RV571.GetState_AI();
RV571(bSetStatusOnAutomatic := bSetStatusOn_RV500,
	fSetPointAutomatic := fSetPoint,
	bAlgorithmPermission := bAlgorithmPermission,
	fTemperatureExternal := fMeanHallTemperature,
	nControlModeAutomatic := nControlMode_RV500);
RV571.SetState_AO();

RV572.GetState_AI();
RV572(bSetStatusOnAutomatic := bSetStatusOn_RV500,
	fSetPointAutomatic := fSetPoint,
	bAlgorithmPermission := bAlgorithmPermission,
	fTemperatureExternal := fMeanHallTemperature,
	nControlModeAutomatic := nControlMode_RV500);
RV572.SetState_AO();

RV573.GetState_AI();
RV573(bSetStatusOnAutomatic := bSetStatusOn_RV500,
	fSetPointAutomatic := fSetPoint,
	bAlgorithmPermission := bAlgorithmPermission,
	fTemperatureExternal := fMeanHallTemperature,
	nControlModeAutomatic := nControlMode_RV500);
RV573.SetState_AO();

//sensors
PS500();
PS500.GetState_AI();
TS541();
TS541.GetState_AI();
TS542();
TS542.GetState_AI();
TS543();
TS543.GetState_AI();
TS551();
TS551.GetState_AI();
TS552();
TS552.GetState_AI();
TS553();
TS553.GetState_AI();
TS561();
TS561.GetState_AI();
TS562();
TS562.GetState_AI();
TS563();
TS563.GetState_AI();
TS571();
TS571.GetState_AI();
TS572();
TS572.GetState_AI();
TS573();
TS573.GetState_AI();

WMZ405(aHeatCounterTelegramm := aTelegramm_WMZ405);

METHOD CalculateAverageTemperature : REAL
VAR_INPUT
	fActualTemperature : REAL;
END_VAR
VAR_OUTPUT
	fMeanTemperature : REAL;
END_VAR
VAR_INST
	fTemperature_init : REAL;
	fMinutes_Moving_Average : UINT := 2;
	
	stParameters_Average_Temperature : ST_CTRL_MOVING_AVERAGE_PARAMS;
	aHallTemperatureBuffer 				: ARRAY [1..360] OF FLOAT := [360(15)];
END_VAR
//fTemperature_init := 

stParameters_Average_Temperature.tCtrlCycleTime := T#1S;
stParameters_Average_Temperature.tTaskCycleTime := GlobalVariables.tTaskCycleTime_MAIN;
stParameters_Average_Temperature.nSamplesToFilter := fMinutes_Moving_Average*60; (* 1min= 60 sec*)
stParameters_Average_Temperature.pWorkArray_ADR := ADR(aHallTemperatureBuffer);
stParameters_Average_Temperature.nWorkArray_SIZEOF := SIZEOF(aHallTemperatureBuffer);

Moving_Average_Hall_Temperature(
	fIn := fActualTemperature,
	fManSyncValue := 15,
	bSync := FALSE,
	eMode := 2,
	bHold := FALSE,
	stParams := stParameters_Average_Temperature);
fMeanTemperature := LREAL_TO_REAL(Moving_Average_Hall_Temperature.fOut);
END_METHOD

METHOD PROTECTED  CheckError : BOOL
VAR_INPUT
END_VAR
VAR_OUTPUT
	bError : BOOL;
END_VAR
VAR
	bError_PU405 : BOOL;
	bError_PU500 : BOOL;
END_VAR
//check pumps for errors
bError_PU405 := PU405.bError;
bError_PU500 := PU500.bError;

bError := bError_PU405 OR bError_PU500;
END_METHOD

METHOD PRIVATE LocalControl : BOOL
VAR_INPUT
END_VAR
VAR
END_VAR
CharacteristicCurve_Parameters.fAmbientTempMax := localDefaultParameters.aLimitsAmbientTemperature[2];
CharacteristicCurve_Parameters.fAmbientTempMin := localDefaultParameters.aLimitsAmbientTemperature[1];
CharacteristicCurve_Parameters.fForeRunTempMax := localDefaultParameters.aLimitsFeedTemperature[1];
CharacteristicCurve_Parameters.fForeRunTempMin := localDefaultParameters.aLimitsFeedTemperature[2];
CharacteristicCurve_Parameters.tCtrlCycleTime := GlobalVariables.tCtrlCycleTime_MAIN;
CharacteristicCurve_Parameters.tTaskCycleTime := GlobalVariables.tTaskCycleTime_MAIN;

CharacteristicCurve(fAmbientTemperature := stAmbientState.fOutsideTemperature,
	fOffsetTemperature := 0,
	bLimitFlowTemp := TRUE,
	stParams := CharacteristicCurve_Parameters);
fSetPoint_RV500 := LREAL_TO_REAL(CharacteristicCurve.fOut);
	
IF bHeatingMode THEN
	nControlMode_RV500 := 1;
ELSE
	nControlMode_RV500 := 2;	
END_IF
END_METHOD

METHOD PROTECTED  Operational : BOOL
VAR_INPUT
END_VAR
VAR_OUTPUT
	bSwitchToWorking : BOOL := FALSE;
END_VAR
bSetStatusOn_RV500 := TRUE;
bSetStatusOn_PU405 := TRUE;
bSetStatusOn_PU500 := TRUE;

IF PU405.bStatusOn AND PU500.bStatusOn THEN
	bSwitchToWorking := TRUE;
END_IF
END_METHOD

METHOD PROTECTED  RampDown : BOOL
VAR_INPUT
END_VAR
VAR_OUTPUT
	bRampDownFinished : BOOL := FALSE;
END_VAR
bSetStatusOn_PU405 := FALSE;
bSetStatusOn_PU500 := FALSE;
bSetStatusOn_RV500 := FALSE;
bSetStatusOn_SV_HNLT := FALSE;
bSetStatusOn_SV_CN := FALSE;
	
IF SV_HNLT.localState.nPosition=2 AND SV_HNLT.localState.nPosition=2 AND SV_CN.localState.nPosition=2 AND SV_CN.localState.nPosition=2 THEN
	bRampDownFinished := TRUE;		
END_IF
END_METHOD

METHOD PROTECTED  RampUp : BOOL
VAR_INPUT
END_VAR
VAR_OUTPUT
	bRampUpFinished : BOOL := FALSE;
END_VAR
IF bHeatingMode THEN
	bSetStatusOn_SV_HNLT := TRUE;
	bSetStatusOn_SV_CN := FALSE;
	IF SV_HNLT.localState.nPosition=3 AND SV_HNLT.localState.nPosition=3 AND SV_CN.localState.nPosition=2 AND SV_CN.localState.nPosition=2 THEN
		bRampUpFinished := TRUE;		
	END_IF	
ELSE
	bSetStatusOn_SV_HNLT := FALSE;
	bSetStatusOn_SV_CN := TRUE;
	IF SV_HNLT.localState.nPosition=2 AND SV_HNLT.localState.nPosition=2 AND SV_CN.localState.nPosition=3 AND SV_CN.localState.nPosition=3 THEN
		bRampUpFinished := TRUE;		
	END_IF	
END_IF
END_METHOD

METHOD PRIVATE SelectLocalControlMode : BOOL
VAR_INPUT
END_VAR
IF control.bManualModeActivated THEN
	bHeatingMode := localSetParameters.bHeatingModeManual;
ELSIF control.bAlgorithmModeActivated AND bAlgorithmPermission THEN
	bHeatingMode := localSetParameters.bHeatingModeAlgorithm;
ELSE
	bHeatingMode := bHeatingModeAutomatic;
END_IF
END_METHOD

METHOD PROTECTED   SetSetPointLimits : BOOL
VAR_INPUT
END_VAR
aSetPointLimits[1] := localDefaultParameters.aSetPointLimitsTemperature[1];
aSetPointLimits[2] := localDefaultParameters.aSetPointLimitsTemperature[2];
END_METHOD

METHOD PROTECTED  SetState : BOOL
VAR_INPUT
END_VAR
VAR_OUTPUT
END_VAR
fOperatingPoint := stAmbientState.fHallTemperature;

controlState.bStatusOn := bSetStatusOn;
setPointState.aSetPointLimits := aSetPointLimits;
setPointState.fSetPoint := fSetPoint;
setPointState.fOperatingPoint := fOperatingPoint;
setPointState.sSetPointUnit := 'degreeC';
setPointState.sOperatingPointUnit := 'degreeC';
END_METHOD

METHOD PRIVATE SwitchMode : BOOL
VAR_INPUT
	bSwitchToHeating : BOOL; //if false switch to cooling
END_VAR
VAR_OUTPUT
	bFinishedSwitchMode : BOOL := FALSE;
END_VAR
VAR_INST
	bRampDownFinished : BOOL := FALSE;
END_VAR
//check system state
IF bRampDownFinished THEN
	IF bSwitchToHeating THEN
		//close valve in cooling network
		bSetStatusOn_SV_CN := FALSE;	
		IF SV_CN.localState.nPosition=2 AND SV_CN.localState.nPosition=2 THEN
			bSetStatusOn_SV_HNLT := TRUE;	
		END_IF

		IF SV_HNLT.localState.nPosition=3 AND SV_HNLT.localState.nPosition=3 THEN
			//reset instant variable and switch on pump
			bRampDownFinished := FALSE;			
			bFinishedSwitchMode := TRUE;
			bSetStatusOn_PU405 := TRUE;
		END_IF
		
	ELSE
		//close valve in heating network
		bSetStatusOn_SV_HNLT := FALSE;
		//wait until valves in heating network are closed before opening valves in cooling network
		IF SV_HNLT.localState.nPosition=2 AND SV_HNLT.localState.nPosition=2 THEN
			bSetStatusOn_SV_CN := TRUE;
		END_IF
		IF SV_CN.localState.nPosition=3 AND SV_CN.localState.nPosition=3 THEN
			//reset instant variable and switch on pump
			bRampDownFinished := FALSE;			
			bFinishedSwitchMode := TRUE;
			bSetStatusOn_PU405 := TRUE;	
		END_IF
	END_IF
ELSE
	bSetStatusOn_PU405 := FALSE;
	IF NOT PU405.bStatusOn THEN
		bRampDownFinished := TRUE;
	END_IF
END_IF
END_METHOD

METHOD PROTECTED  Working : BOOL
VAR_INPUT
END_VAR
VAR_OUTPUT
	bSwitchToOperational : BOOL := FALSE;
END_VAR
//empty method
END_METHOD

END_FUNCTION_BLOCK

// ---- POUs/04 Systems/LinkageSystems/FB_UnderfloorHeatingSystem.TcPOU
FUNCTION_BLOCK FB_UnderfloorHeatingSystem EXTENDS FB_SystemContinous
VAR_INPUT
	bHeatingModeAutomatic : BOOL; //control mode: 0 = heating mode, 1 = cooling mode
	stAmbientState : ST_AmbientState;
END_VAR
VAR_OUTPUT
END_VAR
VAR
	{attribute 'OPC.UA.DA' := '1'}
	localSetParameters : ST_UnderfloorHeatingSetParameters;

	//default parameters
	localDefaultParameters : ST_UnderfloorHeatingDefaultParameters;	
	
	//pumps
	stPU425DefaultParameters : ST_PumpGrundfosMagna3DefaultParameters;
	PU425 : FB_PumpGrundfosMagna3 := (ST_DefaultParameters := stPU425DefaultParameters);	
	
	//valves
	stSV423DefaultParameters : ST_DiscreteValveDefaultParameters := (nFeedback := 3);
	stSV424DefaultParameters : ST_DiscreteValveDefaultParameters := (nFeedback := 3);
	stRV425DefaultParameters : ST_MixingValveDefaultParameters := (bFeedbackSignal := FALSE, tTaskCycleTime := GlobalVariables.tTaskCycleTime_MAIN, tCtrlCycleTime := GlobalVariables.tCtrlCycleTime_MAIN);	
	
	SV423 : FB_DiscreteValve := (ST_DefaultParameters := stSV423DefaultParameters); 
	SV424 : FB_DiscreteValve := (ST_DefaultParameters := stSV424DefaultParameters);
	RV425 : FB_MixingValve := (ST_DefaultParameters := stRV425DefaultParameters);
	WMZ425 : FB_MollineEHeatCounter;
	
	//internal variables
	bHeatingMode 			: BOOL;
	bSetStatusOn_PU425 		: BOOL;
	bSetStatusOn_SV423		: BOOL;
	bSetStatusOn_SV424		: BOOL;
	bSetStatusOn_RV425 		: BOOL;
	fSetPoint_Internal 		: REAL;
	nControlMode_RV425 		: E_MixingValveControlMode; 	
	
	//characteristic curves and controllers
	CharacteristicCurve 			: FB_CTRL_FLOW_TEMP_SETPOINT_GEN;
	CharacteristicCurve_Parameters	: ST_CTRL_FLOW_TEMP_SETPOINT_GEN_PARAMS;
	
	//triggers
	SwitchToHeating : R_TRIG;
	SwitchToCooling : F_TRIG;
	bFinishedSwitchMode : BOOL := TRUE;
END_VAR

//check if heating mode has switched
SelectLocalControlMode();
LocalControl();
fSetPointAutomatic := fSetPoint_Internal;
SwitchToHeating(CLK := bHeatingMode);
SwitchToCooling(CLK := bHeatingMode);

//MAIN must be called before SwitchMode to prevent pump signal chattering (signal is written after SwitchMode function), SwitchMode may only be called if system is on
MAIN();

//disrupt calling SystemFlowControl via MAIN() when mode is switched and call SwitchMode()
IF ((SwitchToHeating.Q OR SwitchToCooling.Q) OR NOT bFinishedSwitchMode) AND bSetStatusOn THEN
	SwitchMode(bSwitchToHeating := bHeatingMode,
		bFinishedSwitchMode => bFinishedSwitchMode);
END_IF;

//pumps
PU425.GetState_Profibus();
PU425(bSetStatusOnAutomatic := bSetStatusOn_PU425,
	fSetPointAutomatic := 100,
	bAlgorithmPermission := bAlgorithmPermission,
	nControlModeAutomatic := 0);
PU425.SetState_Profibus();

//valves in thermal networks
RV425.GetState_AI();
RV425(bSetStatusOnAutomatic := bSetStatusOn_RV425,
	fSetPointAutomatic := fSetPoint_Internal,
	bAlgorithmPermission := bAlgorithmPermission,
	fTemperatureExternal := PU425.fTemperatureInternal,
	fThermalPowerExternal := WMZ425.fHeatFlowRate,
	nControlModeAutomatic := nControlMode_RV425);
RV425.SetState_AO();

SV423.GetState_BI();
SV423(bSetStatusOnAutomatic := bSetStatusOn_SV423,
	bAlgorithmPermission := bAlgorithmPermission);
SV423.SetState_BO();

SV424.GetState_BI();
SV424(bSetStatusOnAutomatic := bSetStatusOn_SV423,
	bAlgorithmPermission := bAlgorithmPermission);
SV424.SetState_BO();

WMZ425(aHeatCounterTelegramm := aTelegramm_WMZ425);

METHOD PROTECTED  CheckError : BOOL
VAR_INPUT
END_VAR
VAR_OUTPUT
	bError : BOOL;
END_VAR
VAR
END_VAR
//check pumps for errors
bError :=  PU425.bError;
END_METHOD

METHOD PRIVATE LocalControl : BOOL
VAR_INPUT
END_VAR
VAR
END_VAR
CharacteristicCurve_Parameters.fAmbientTempMax := localDefaultParameters.aLimitsAmbientTemperature[2];
CharacteristicCurve_Parameters.fAmbientTempMin := localDefaultParameters.aLimitsAmbientTemperature[1];
CharacteristicCurve_Parameters.fForeRunTempMax := localDefaultParameters.aLimitsFeedTemperature[1];
CharacteristicCurve_Parameters.fForeRunTempMin := localDefaultParameters.aLimitsFeedTemperature[2];
CharacteristicCurve_Parameters.tCtrlCycleTime := GlobalVariables.tCtrlCycleTime_MAIN;
CharacteristicCurve_Parameters.tTaskCycleTime := GlobalVariables.tTaskCycleTime_MAIN;

CharacteristicCurve(fAmbientTemperature := stAmbientState.fOutsideTemperature,
	fOffsetTemperature := 0,
	bLimitFlowTemp := TRUE,
	stParams := CharacteristicCurve_Parameters);
fSetPoint_Internal := LREAL_TO_REAL(CharacteristicCurve.fOut);
	
IF bHeatingMode THEN
	nControlMode_RV425 := 1;
ELSE
	nControlMode_RV425 := 2;	
END_IF
END_METHOD

METHOD PROTECTED  Operational : BOOL
VAR_INPUT
END_VAR
VAR_OUTPUT
	bSwitchToWorking : BOOL := FALSE;
END_VAR
bSetStatusOn_RV425 := TRUE;
bSetStatusOn_PU425 := TRUE;

IF PU425.bStatusOn THEN
	bSwitchToWorking := TRUE;
END_IF
END_METHOD

METHOD PROTECTED  RampDown : BOOL
VAR_INPUT
END_VAR
VAR_OUTPUT
	bRampDownFinished : BOOL := FALSE;
END_VAR
bSetStatusOn_PU425 := FALSE;
bSetStatusOn_RV425 := FALSE;
	
IF PU425.bStatusOn THEN
	bRampDownFinished := TRUE;		
END_IF
END_METHOD

METHOD PROTECTED  RampUp : BOOL
VAR_INPUT
END_VAR
VAR_OUTPUT
	bRampUpFinished : BOOL := FALSE;
END_VAR
IF bHeatingMode THEN
	//bSetStatusOn_SV423 := FALSE;
	//bSetStatusOn_SV424 := FALSE;
	IF SV423.localState.nPosition=3 AND SV424.localState.nPosition=3 THEN
		bRampUpFinished := TRUE;		
	END_IF	
ELSE
	//bSetStatusOn_SV423 := TRUE;
	//bSetStatusOn_SV424 := TRUE;
	IF SV423.localState.nPosition=2 AND SV424.localState.nPosition=2 THEN
		bRampUpFinished := TRUE;		
	END_IF	
END_IF
END_METHOD

METHOD PRIVATE SelectLocalControlMode : BOOL
VAR_INPUT
END_VAR
IF control.bManualModeActivated THEN
	bHeatingMode := localSetParameters.bHeatingModeManual;
ELSIF control.bAlgorithmModeActivated AND bAlgorithmPermission THEN
	bHeatingMode := localSetParameters.bHeatingModeAlgorithm;
ELSE
	bHeatingMode := bHeatingModeAutomatic;
END_IF
END_METHOD

METHOD PROTECTED   SetSetPointLimits : BOOL
VAR_INPUT
END_VAR
aSetPointLimits[1] := localDefaultParameters.aSetPointLimitsTemperature[1];
aSetPointLimits[2] := localDefaultParameters.aSetPointLimitsTemperature[2];
END_METHOD

METHOD PROTECTED  SetState : BOOL
VAR_INPUT
END_VAR
VAR_OUTPUT
END_VAR
fOperatingPoint := PU425.fTemperatureInternal;

controlState.bStatusOn := bSetStatusOn;
setPointState.aSetPointLimits := aSetPointLimits;
setPointState.fSetPoint := fSetPoint;
setPointState.fOperatingPoint := fOperatingPoint;
setPointState.sSetPointUnit := 'degreeC';
setPointState.sOperatingPointUnit := 'degreeC';
END_METHOD

METHOD PRIVATE SwitchMode : BOOL
VAR_INPUT
	bSwitchToHeating : BOOL; //if false switch to cooling
END_VAR
VAR_OUTPUT
	bFinishedSwitchMode : BOOL := FALSE;
END_VAR
VAR_INST
	bRampDownFinished : BOOL := FALSE;
END_VAR
//check system state
IF bRampDownFinished THEN
	IF bSwitchToHeating THEN
		//false - valve connects heating network
		bSetStatusOn_SV423 := FALSE;
		bSetStatusOn_SV424 := FALSE;	

		IF SV423.localState.nPosition=3 AND SV424.localState.nPosition=3 THEN
			//reset instant variable and switch on pump
			bRampDownFinished := FALSE;			
			bFinishedSwitchMode := TRUE;
			bSetStatusOn_PU425 := TRUE;
		END_IF
		
	ELSE
		//true - connects cooling network
		bSetStatusOn_SV423 := TRUE;
		bSetStatusOn_SV424 := TRUE;	

		IF SV423.localState.nPosition=2 AND SV424.localState.nPosition=2 THEN
			//reset instant variable and switch on pump
			bRampDownFinished := FALSE;			
			bFinishedSwitchMode := TRUE;
			bSetStatusOn_PU425 := TRUE;
		END_IF
	END_IF
ELSE
	bSetStatusOn_PU425 := FALSE;
	IF NOT PU425.bStatusOn THEN
		bRampDownFinished := TRUE;
	END_IF
END_IF
END_METHOD

METHOD PROTECTED  Working : BOOL
VAR_INPUT
END_VAR
VAR_OUTPUT
	bSwitchToOperational : BOOL := FALSE;
END_VAR
//empty method
END_METHOD

END_FUNCTION_BLOCK

// ---- POUs/05 Thermal Networks/FB_HnhtCnLinkage.TcPOU
FUNCTION_BLOCK FB_HnhtCnLinkage
VAR_INPUT	
	//control struct for hnht cn linkage
	controlAutomatic : ST_HnhtCnLinkageControl;
END_VAR
VAR_OUTPUT
END_VAR
VAR
	//systems
	VentilationSystem : FB_VentilationSystem;
	
	//internal variables
	bAlgorithmPermission : BOOL;
	
	//PCM Supply System
	PCMSupplySystem : FB_PCMSupplySystem;
END_VAR

bAlgorithmPermission := controlAutomatic.bAlgorithmPermission_HNHT AND controlAutomatic.bAlgorithmPermission_CN;

//ventilation system has its own controller, only valves are controlled
VentilationSystem(bSetStatusOnAutomatic := TRUE,
	fSetPointAutomatic := 0,
	bAlgorithmPermission := bAlgorithmPermission,
	bHeatingModeAutomatic := controlAutomatic.bHeatingMode);

PCMSupplySystem(bSetStatusOnAutomatic := TRUE, 
	bAlgorithmPermission := bAlgorithmPermission,
	fSetPointAutomatic := 9);

END_FUNCTION_BLOCK

// ---- POUs/04 Systems/LinkageSystems/FB_VentilationSystem.TcPOU
FUNCTION_BLOCK FB_VentilationSystem EXTENDS FB_SystemContinous
VAR_INPUT
	bHeatingModeAutomatic : BOOL; //control mode: 0 = heating mode, 1 = cooling mode
END_VAR
VAR_OUTPUT
END_VAR
VAR
	{attribute 'OPC.UA.DA' := '1'}
	localSetParameters : ST_VentilationSetParameters;
	
	localDefaultParameters : ST_VentilationDefaultParameters;
	
	//valves
	stSV453DefaultParameters : ST_DiscreteValveDefaultParameters := (nFeedback := 3);
	stSV454DefaultParameters : ST_DiscreteValveDefaultParameters := (nFeedback := 3);
	SV453 : FB_DiscreteValve := (ST_DefaultParameters := stSV453DefaultParameters);
	SV454 : FB_DiscreteValve := (ST_DefaultParameters := stSV454DefaultParameters);
	
	//pump (pump is just read)
	stPU455DefaultParameters : ST_PumpGrundfosMagna3DefaultParameters := (tTaskCycleTime := GlobalVariables.tTaskCycleTime_MAIN, tCtrlCycleTime := GlobalVariables.tCtrlCycleTime_MAIN);
	PU455 : FB_PumpGrundfosMagna3 := (ST_DefaultParameters := stPU455DefaultParameters);
	
	WMZ455 : FB_MollineEHeatCounter;
	
	//ventilation 
	//Ventilation : FB_Ventilation; //commented out for merge in dev, as modbus write needs to be deactivated before bugs are fixed
	
	//electricity meter
	EM45x : FB_JanitzaSensor;
	
	
	
	bHeatingMode 			: BOOL;
	bSetStatusOn_SV453		: BOOL;
	bSetStatusOn_SV454		: BOOL;
END_VAR

SelectLocalControlMode();
MAIN();
(* Ventilation.GetState();
Ventilation(
	fSetPointAutomatic := fSetPoint,
	bSetStatusOnAutomatic := FALSE,
	bAlgorithmPermission := bAlgorithmPermission,
	sIPAddress := GlobalVariables.sIP_Ventilation);
Ventilation.SetState();
EM45x(
	sIPAddress := GlobalVariables.sIP_Janitza_Ventilation);  

*)

IF bHeatingMode THEN
	bSetStatusOn_SV453 := TRUE;
	bSetStatusOn_SV454 := TRUE;
ELSE
	bSetStatusOn_SV453 := FALSE;
	bSetStatusOn_SV454 := FALSE;
END_IF

SV453.GetState_BI();
SV453(bSetStatusOnAutomatic := bSetStatusOn_SV453,
	bAlgorithmPermission := bAlgorithmPermission);
SV453.SetState_BO();

SV454.GetState_BI();
SV454(bSetStatusOnAutomatic := bSetStatusOn_SV454,
	bAlgorithmPermission := bAlgorithmPermission);
SV454.SetState_BO();


	
	
	
	

//PU455 and RV455 is controlled by ventilation unit
PU455.GetState_Profibus();
PU455();

WMZ455(aHeatCounterTelegramm := aTelegramm_WMZ455);

METHOD PROTECTED  CheckError : BOOL
VAR_INPUT
END_VAR
VAR_OUTPUT
	bError : BOOL;
END_VAR
IF (SV453.localState.nPosition = 2 AND SV454.localState.nPosition = 3) OR (SV453.localState.nPosition = 3 AND SV454.localState.nPosition = 2) THEN
	bError := TRUE;
ELSE
	bError := FALSE;
END_IF
END_METHOD

METHOD PROTECTED  Operational : BOOL
VAR_INPUT
END_VAR
VAR_OUTPUT
	bSwitchToWorking : BOOL := FALSE;
END_VAR
//empty
END_METHOD

METHOD PROTECTED  RampDown : BOOL
VAR_INPUT
END_VAR
VAR_OUTPUT
	bRampDownFinished : BOOL := FALSE;
END_VAR
//empty
END_METHOD

METHOD PROTECTED  RampUp : BOOL
VAR_INPUT
END_VAR
VAR_OUTPUT
	bRampUpFinished : BOOL := FALSE;
END_VAR
//empty
END_METHOD

METHOD PRIVATE SelectLocalControlMode : BOOL
VAR_INPUT
END_VAR
IF control.bManualModeActivated THEN
	bHeatingMode := localSetParameters.bHeatingModeManual;
ELSIF control.bAlgorithmModeActivated AND bAlgorithmPermission THEN
	bHeatingMode := localSetParameters.bHeatingModeAlgorithm;
ELSE
	bHeatingMode := bHeatingModeAutomatic;
END_IF
END_METHOD

METHOD PROTECTED   SetSetPointLimits : BOOL
VAR_INPUT
END_VAR
aSetPointLimits[1] := localDefaultParameters.aSetPointLimitsTemperature[1];
aSetPointLimits[2] := localDefaultParameters.aSetPointLimitsTemperature[2];
END_METHOD

METHOD PROTECTED  SetState : BOOL
VAR_INPUT
END_VAR
VAR_OUTPUT
END_VAR
fOperatingPoint := 0;

controlState.bStatusOn := bSetStatusOn;
setPointState.aSetPointLimits := aSetPointLimits;
setPointState.fSetPoint := 0;
setPointState.fOperatingPoint := fOperatingPoint;
setPointState.sSetPointUnit := '-';
setPointState.sOperatingPointUnit := '-';
END_METHOD

METHOD PROTECTED  Working : BOOL
VAR_INPUT
END_VAR
VAR_OUTPUT
	bSwitchToOperational : BOOL := FALSE;
END_VAR
//empty
END_METHOD

END_FUNCTION_BLOCK

// ---- POUs/02 Sensors/FB_JanitzaSensor.TcPOU
FUNCTION_BLOCK FB_JanitzaSensor
VAR_INPUT
	sIPAddress : STRING(15);
END_VAR
VAR_OUTPUT
	fPower : REAL; //measured power in watt
	bError : BOOL; 
	nErrID : UDINT; 
END_VAR
VAR
	
	{attribute 'OPC.UA.DA' := '1'}
	sensorState : ST_JanitzaState;
	//modbus tcp communication
	ModbusReader_19026 : FB_MBReadInputRegs; //read reg 19026 (power (W) ventilation)
	
	//define array to store data from every ModbusReader
	aModbus_19026 : ARRAY [0..1] OF WORD;
	
	//modbus timer
	bReadModbus	: BOOL := FALSE;
	bStartTimer : BOOL;
	Timer : TON;
	
	bAwaitData : BOOL; //mark: Results of this still pending
	aTmp : ARRAY[0..1] OF WORD; //temp. buffer for byte-swap (won't overwrite the original)
	
END_VAR

//Start and check timer for 2s interval
Timer(IN := bStartTimer,
	PT := T#2S);
	
bStartTimer := TRUE;
IF Timer.Q THEN
	bReadModbus := TRUE;
	bStartTimer := FALSE;	
	bAwaitData := TRUE; // we expecting a answer
END_IF

ModbusReader_19026(
	sIPAddr := sIPAddress,
	nTCPPort := 502,
	nUnitID := 32,
	nQuantity := 2,
	nMBAddr := 19026 + 32768,
	cbLength := 4,
	pDestAddr := ADR(aModbus_19026),
	bExecute := bReadModbus,
	tTimeout  := T#20S);
	
bReadModbus := FALSE;
	
bError := ModbusReader_19026.bError;
nErrID := ModbusReader_19026.nErrId; 

IF bAwaitData AND NOT ModbusReader_19026.bBusy AND NOT ModbusReader_19026.bError THEN
	bAwaitData := FALSE; 
    // Byte-Swap for every WORD (51794 = 19026+32768: Word sequence is LE, But the Bytes in the Word are BE)
    aModbus_19026[0] := SHL(aModbus_19026[0] AND 16#00FF, 8) OR SHR(aModbus_19026[0] AND 16#FF00, 8);
    aModbus_19026[1] := SHL(aModbus_19026[1] AND 16#00FF, 8) OR SHR(aModbus_19026[1] AND 16#FF00, 8);
	MEMCPY(ADR(fPower), ADR(aModbus_19026), SIZEOF(fPower));
	bStartTimer := TRUE; 
END_IF

//sensor state
sensorState.fPower := fPower/1000;
sensorState.sPowerUnit := 'kW';

END_FUNCTION_BLOCK

// ---- POUs/04 Systems/CoolingSystems/FB_PCMSupplySystem.TcPOU
FUNCTION_BLOCK FB_PCMSupplySystem EXTENDS FB_SystemContinous
VAR_INPUT
	nControlModeAutomatic : E_PCMSystemControlMode;
	
END_VAR
VAR_OUTPUT
END_VAR
VAR
	
	{attribute 'OPC.UA.DA' := '1'}
	localSetParameters : ST_PCMSystemSetParameters;
	
	//heat meters
	WMZ900 : FB_MollineUltramess403HeatCounter; //pcm storage
	WMZ935 : FB_MollineUltramess403HeatCounter; //chiller
	
	//temperature sensors
	
	TS901 : FB_TemperatureSensor_KL3214;
	TS902 : FB_TemperatureSensor_KL3214;
	TS903 : FB_TemperatureSensor_KL3214;
	TS910 : FB_TemperatureSensor_KL3214;
	TS911 : FB_TemperatureSensor_KL3214;
	TS950 : FB_TemperatureSensor_KL3214;
	TS951 : FB_TemperatureSensor_KL3214;
	
	//valves
	ST_RV950DefaultParameters : ST_MixingValveDefaultParameters := (bFeedbackSignal := FALSE, tTaskCycleTime := GlobalVariables.tTaskCycleTime_MAIN, tCtrlCycleTime := GlobalVariables.tCtrlCycleTime_MAIN);
	RV950 : FB_MixingValve := (ST_DefaultParameters := ST_RV950DefaultParameters);
	
	// pcm chiller
	PCMChiller : FB_PCMChiller;
	
	// PCMStorage
	PCMStorage : FB_PCMStorage;
	
	//internal variables
	nControlMode : E_PCMSystemControlMode;
	
	bSetStatusOn_RV950 : BOOL; 
	
	
END_VAR

SelectLocalControlMode();


WMZ900(aHeatCounterTelegramm := aTelegramm_WMZ900);
WMZ935(aHeatCounterTelegramm := aTelegramm_WMZ935);
	
TS901();
TS901.GetState_AI();
TS902();
TS902.GetState_AI();
TS903();
TS903.GetState_AI();
TS910();
TS910.GetState_AI();
TS911();
TS911.GetState_AI();
TS950();
TS950.GetState_AI();
TS951();
TS951.GetState_AI();

RV950.GetState_AI();
RV950(bSetStatusOnAutomatic := bSetStatusOn_RV950,
	fSetPointAutomatic := 100,
	bAlgorithmPermission := TRUE,
	fTemperatureExternal := TS950.fTemperature,
	nControlModeAutomatic := 0);
RV950.SetState_AO();

PCMChiller.GetState(); 
PCMChiller(bSetStatusOnAutomatic := FALSE, 
	bAlgorithmPermission := bAlgorithmPermission,
	fSetPointAutomatic := fSetPoint);
PCMChiller.SetState();

METHOD PROTECTED  CheckError : BOOL
VAR_INPUT
END_VAR
VAR_OUTPUT
	bError : BOOL;
END_VAR
END_METHOD

METHOD LocalControl : BOOL
VAR_INPUT
	
END_VAR
CASE nControlMode OF
	0: //stand-by
	PCMChiller.bStatusOn := FALSE; 
	 	
	1: //direct cooling 
	PCMChiller.nControlModeAutomatic := 0; 
	PCMChiller.fSetPointAutomatic := fSetPoint; 
	bSetStatusOn_RV950 := FALSE; 
	
	2: //charge pcm
	PCMChiller.nControlModeAutomatic := 0; 
	PCMChiller.fSetPointAutomatic := fSetPoint;
	bSetStatusOn_RV950 := TRUE; 
	
	3: //discharge pcm
	PCMChiller.nControlModeAutomatic := 1; 
	bSetStatusOn_RV950 := TRUE; 
		
END_CASE
END_METHOD

METHOD PROTECTED  Operational : BOOL
VAR_INPUT
END_VAR
VAR_OUTPUT
	bSwitchToWorking : BOOL := FALSE;
END_VAR
END_METHOD

METHOD PROTECTED  RampDown : BOOL
VAR_INPUT
END_VAR
VAR_OUTPUT
	bRampDownFinished : BOOL := FALSE;
END_VAR
END_METHOD

METHOD PROTECTED  RampUp : BOOL
VAR_INPUT
END_VAR
VAR_OUTPUT
	bRampUpFinished : BOOL := TRUE;
END_VAR
END_METHOD

METHOD SelectLocalControlMode : BOOL
VAR_INPUT
END_VAR
IF control.bManualModeActivated THEN
	nControlMode := localSetParameters.nControlModeManual;
ELSIF control.bAlgorithmModeActivated AND bAlgorithmPermission THEN
	nControlMode := localSetParameters.nControlModeAlgorithm;
ELSE
	nControlMode := nControlModeAutomatic;
END_IF
END_METHOD

METHOD PROTECTED   SetSetPointLimits : BOOL
VAR_INPUT
END_VAR
END_METHOD

METHOD PROTECTED  SetState : BOOL
VAR_INPUT
END_VAR
VAR_OUTPUT
END_VAR
END_METHOD

METHOD PROTECTED  Working : BOOL
VAR_INPUT
END_VAR
VAR_OUTPUT
	bSwitchToOperational : BOOL := FALSE;
END_VAR
//Implementing different control modes (next time)
END_METHOD

END_FUNCTION_BLOCK

// ---- POUs/01 Actuators/CoolingUnits/FB_PCMChiller.TcPOU
FUNCTION_BLOCK FB_PCMChiller EXTENDS FB_ActuatorContinous
VAR_INPUT
	fExternalTemperature : REAL; 
	nControlModeAutomatic : E_PCMControlMode;
END_VAR
VAR_OUTPUT
END_VAR
VAR
	
	{attribute 'OPC.UA.DA' := '1'}
	localState : ST_pcmChillerState;
	//default parameters
	localDefaultParameters : ST_pcmChillerDefaultParameters;
	//I/O Links
	nRemoteControl_OUT AT %Q* : DINT;
	nSetPointMediumTemperature_OUT AT %Q* : LREAL;
	fAmbientTemperature_IN AT %I* : LREAL;
	fMediumOutletTemperature_IN AT %I* : LREAL; 
	fCoolingCapacity_IN AT %I* : DINT; 
	fCoolingEER_IN AT %I* : LREAL; 
	fFlowValue_IN AT %I* : LREAL; 
	fFanValue_IN AT %I* : DINT; 
	fCompressorSpeed_IN AT %I* : DINT; 
	fEEVValue_IN AT %I* : LREAL; 
	fEEVPosition_IN AT %I* : DINT; 
	fInputPower_IN AT %I* : DINT; 
	fEnvironmentTemperature_IN AT %I* : LREAL;
	
	//internal variables
	nControlMode : E_PCMControlMode;
END_VAR

MAIN();

METHOD GetState : BOOL
VAR_INPUT
END_VAR
//control state


//setpoint state
setPointState.fOperatingPoint := fExternalTemperature; //adjust fExternalTemperature to the right variable
setPointState.sOperatingPointUnit := 'degreeC'; 
fOperatingPoint := fExternalTemperature; 

//local state
localState.fAmbientTemperature := fAmbientTemperature_IN;
localState.fCompressorSpeed := fCompressorSpeed_IN;
localState.fCoolingCapacity := fCoolingCapacity_IN; 
localState.fCoolingEER := fCoolingEER_IN; 
localState.fEEVPosition := fEEVPosition_IN; 
localState.fEEVValue := fEEVValue_IN; 
localState.fEnvironmentTemperature := fEnvironmentTemperature_IN; 
localState.fFanValue := fFanValue_IN; 
localState.fFlowValue := fFlowValue_IN; 
localState.fInputPower := fInputPower_IN;
localState.fMediumOutletTemperature := fMediumOutletTemperature_IN;
END_METHOD

METHOD PROTECTED  SetSetPointLimits : BOOL
VAR_INPUT
END_VAR
aSetPointLimits[1] := localDefaultParameters.aSetPointLimitsTemperature[1];
aSetPointLimits[2] := localDefaultParameters.aSetPointLimitsTemperature[2];
END_METHOD

METHOD SetState : BOOL
VAR_INPUT
END_VAR
setPointState.fSetPoint := fSetPoint;
setPointState.aSetPointLimits := aSetPointLimits;
setPointState.sSetPointUnit := 'degreeC';


nSetPointMediumTemperature_OUT := fSetPoint;

IF bSetStatusOn THEN
	CASE nControlMode OF
		0: //cooling mode
		nRemoteControl_OUT := 0;
		
		1: //pump mode
		nRemoteControl_OUT := 2;
	END_CASE
ELSE
	nRemoteControl_OUT := 1; //Stand-By
END_IF;
END_METHOD

PROPERTY ST_DefaultParameters : REFERENCE TO ST_pcmChillerDefaultParameters
GET
ST_DefaultParameters REF= localDefaultParameters;
END_GET
SET
localDefaultParameters := ST_DefaultParameters;
END_SET
END_PROPERTY

END_FUNCTION_BLOCK

// ---- POUs/03 Storages/FB_PCMStorage.TcPOU
FUNCTION_BLOCK FB_PCMStorage
VAR_INPUT
END_VAR
VAR_OUTPUT
	{attribute 'OPC.UA.DA' := '1'}
	localState : ST_PCMStorageState;
END_VAR
VAR
	//temperature sensors
	TemperatureSensor : FB_TemperatureSensor_KL3214;
	
	//Temperature
	Temperature: REAL;
	
	// SOC-Value
	SOC_per : REAL; 
	SOC_abs : REAL; 
	
END_VAR

//temperature sensors
TemperatureSensor();
TemperatureSensor.GetState_AI();

Temperature := TemperatureSensor.fTemperature;

CalcSOC(
    Temperature := Temperature, 
    SOC_per => localState.SOCValuePercentage, 
    SOC_abs => localState.SOCValueAbsolute
);

localState.SOCValuePercentage := SOC_per; 
localState.SOCValueAbsolute := SOC_abs; 
localState.TemperatureSensor := Temperature;

METHOD CalcSOC : REAL
VAR_INPUT
	Temperature: REAL;
END_VAR
VAR_OUTPUT
	SOC_per : REAL;
	SOC_abs : REAL;
END_VAR
//derivation and parameter from jonas wendts dissertation
SOC_per := (0.11822542*EXPT(Temperature, 4)-7.4519133*EXPT(Temperature, 3)+174.94045*EXPT(Temperature, 2)-1822.0902*Temperature+7168.3066);

IF SOC_per > 100 THEN
	SOC_per := 100;
ELSIF SOC_per > 100 THEN
	SOC_per := 0; 
END_IF

SOC_abs := (SOC_per/100)*20.43;
END_METHOD

END_FUNCTION_BLOCK

// ---- POUs/05 Thermal Networks/FB_HeatingNetworkLowTemperature.TcPOU
FUNCTION_BLOCK FB_HeatingNetworkLowTemperature
VAR_INPUT
	ambientState : ST_AmbientState;
	
	//control struct for hnlt
	controlAutomatic : ST_HeatingNetworkLowTemperatureControl;	
END_VAR
VAR_OUTPUT
	{attribute 'OPC.UA.DA' := '1'}
	localState : ST_ThermalNetworkState;
END_VAR
VAR
	//systems
	BufferStorage : FB_BufferStorage;
	OuterCapillaryTubeMats : FB_OuterCapillaryTubeMats;
	HVFASystem : FB_HVFAStorageSystem;
	CompressorSystem : FB_CompressorSystem;
	AnnealingOvenSealingSystem : FB_AnnealingOvenSealingSystem;
	DCSystem : FB_DCSystem;
	
	//machines
	AnnealingOvenSealing : FB_AnnealingOven;
	DC : FB_DC;

	//internal variables
	bSetStatusOn_AnnealingOven : BOOL;
	bSetStatusOn_DC : BOOL;
	bError_DC : BOOL;
END_VAR

//buffer storage system
BufferStorage();
localState.fUpperTemperature := BufferStorage.localState.fUpperTemperature;
localState.fMidTemperature := BufferStorage.localState.fMidTemperature;
localState.fLowerTemperature := BufferStorage.localState.fLowerTemperature;
localState.fUpperTemperature_ActiveStorage := HVFASystem.localStorageState.fUpperTemperature;
localState.fLowerTemperature_ActiveStorage := HVFASystem.localStorageState.fLowerTemperature;

//producer
CompressorSystem(bSetStatusOnAutomatic := TRUE,
	bAlgorithmPermission := controlAutomatic.bAlgorithmPermission,
	fSetPointAutomatic := controlAutomatic.fFeedTemperature_Heating);

//consumer
OuterCapillaryTubeMats(bSetStatusOnAutomatic := controlAutomatic.bSetStatusOn_OuterCapillaryTubeMats,
	bAlgorithmPermission := controlAutomatic.bAlgorithmPermission,
	fSetPointAutomatic := controlAutomatic.fFeedTemperature_Cooling,
	stAmbientState := ambientState);
	
AnnealingOvenSealing();
bSetStatusOn_AnnealingOven := AnnealingOvenSealing.bStatusOn_Sealing;
AnnealingOvenSealingSystem(bSetStatusOnAutomatic := bSetStatusOn_AnnealingOven,
	bAlgorithmPermission := controlAutomatic.bAlgorithmPermission,
	fSetPointAutomatic := controlAutomatic.fFeedTemperature_Heating);
	
DC();
bSetStatusOn_DC := (DC.bStatusOn AND NOT DC.bError_Connection);

DCSystem(bSetStatusOnAutomatic := bSetStatusOn_DC,
	bAlgorithmPermission := controlAutomatic.bAlgorithmPermission,
	fSetPointAutomatic := 3); //temperature difference control

//external storages
HVFASystem(bSetStatusOnAutomatic := controlAutomatic.bSetStatusOn_HVFASystem,
	bAlgorithmPermission := controlAutomatic.bAlgorithmPermission,
	fSetPointAutomatic := 70,
	bLoadingAutomatic := controlAutomatic.bLoading_HVFASystem,
	aTelegramm_WMZ7x0 := aTelegramm_WMZ720,
	aTelegramm_WMZx05 := aTelegramm_WMZ205);

END_FUNCTION_BLOCK

// ---- POUs/04 Systems/CoolingSystems/FB_OuterCapillaryTubeMats.TcPOU
FUNCTION_BLOCK FB_OuterCapillaryTubeMats EXTENDS FB_SystemContinous
VAR_INPUT
	stAmbientState : ST_AmbientState;
END_VAR
VAR_OUTPUT
END_VAR
VAR
	//default parameters
	localDefaultParameters : ST_OuterCapillaryTubeMatsDefaultParameters;	
	
	//pumps
	stPU235DefaultParameters : ST_PumpGrundfosMagna3DefaultParameters;
	stPU600DefaultParameters : ST_PumpGrundfosMagna3DefaultParameters;
	
	PU235 : FB_PumpGrundfosMagna3 := (ST_DefaultParameters := stPU235DefaultParameters);
	PU600 : FB_PumpGrundfosMagna3 := (ST_DefaultParameters := stPU600DefaultParameters);	
	PU690 : FB_Pump2Point; //CM pump (storage side)
	
	//valves
	stSV235DefaultParameters : ST_DiscreteValveDefaultParameters := (nFeedback := 0);
	stSV605DefaultParameters : ST_DiscreteValveDefaultParameters := (nFeedback := 3);
	stRV600DefaultParameters : ST_MixingValveDefaultParameters := (bFeedbackSignal := FALSE, tTaskCycleTime := GlobalVariables.tCtrlCycleTime_MAIN, tCtrlCycleTime := GlobalVariables.tCtrlCycleTime_MAIN, fControllerAmplification := 0.012, tControllerIntegralTime := T#36S, fOutMinLimit := 0, fOutMaxLimit := 70);	
	stRV640DefaultParameters : ST_MixingValveDefaultParameters := (bFeedbackSignal := FALSE, tTaskCycleTime := GlobalVariables.tCtrlCycleTime_MAIN, tCtrlCycleTime := GlobalVariables.tCtrlCycleTime_MAIN);
	stRV660DefaultParameters : ST_MixingValveDefaultParameters := (bFeedbackSignal := FALSE, tTaskCycleTime := GlobalVariables.tCtrlCycleTime_MAIN, tCtrlCycleTime := GlobalVariables.tCtrlCycleTime_MAIN);
	
	SV235 : FB_DiscreteValve := (ST_DefaultParameters := stSV235DefaultParameters);
	SV605 : FB_DiscreteValve := (ST_DefaultParameters := stSV605DefaultParameters);
	RV600 : FB_MixingValve := (ST_DefaultParameters := stRV600DefaultParameters);
	RV640 : FB_MixingValve := (ST_DefaultParameters := stRV640DefaultParameters); //east
	RV660 : FB_MixingValve := (ST_DefaultParameters := stRV660DefaultParameters); //west
	
	//sensors
	WMZ235	: FB_MollineC3HeatCounter;
	TS640	: FB_TemperatureSensor; //return temperature east
	TS660 	: FB_TemperatureSensor; //return temperature west
	PS600	: FB_PressureSensor;
	
	//internal variables
	bSetStatusOn_PU235 	: BOOL;
	bSetStatusOn_PU600 	: BOOL;
	bSetStatusOn_PU690 	: BOOL;
	bSetStatusOn_SV235 	: BOOL;	
	bSetStatusOn_RV600 	: BOOL;
	bSetStatusOn_RV640 	: BOOL;
	fSetPoint_RV640 	: REAL;
	bSetStatusOn_RV660 	: BOOL;
	fSetPoint_RV660 	: REAL;
	
	//clock and timer
	stDefaultParameters_Clock : ST_ClockDefaultParameters := (tTaskCycleTime := GlobalVariables.tCtrlCycleTime_MAIN, tCtrlCycleTime := T#1M);
	Clock : FB_Clock := (ST_DefaultParameters := stDefaultParameters_Clock);
	bStartTimer : BOOL;
	Timer : TON;
END_VAR

MAIN();
//use timer because valve has no feedback signal (75 sec)
Timer(IN := bStartTimer,
	PT := T#75S);
Clock();

//pumps
PU235.GetState_Profibus();
PU235(bSetStatusOnAutomatic := bSetStatusOn_PU235,
	fSetPointAutomatic := 70,
	bAlgorithmPermission := bAlgorithmPermission,
	nControlModeAutomatic := 0);
PU235.SetState_Profibus();

//use AUTO-Adapt control mode
PU600.GetState_Profibus();
PU600(bSetStatusOnAutomatic := bSetStatusOn_PU600,
	fSetPointAutomatic := 100,
	bAlgorithmPermission := bAlgorithmPermission,
	nControlModeAutomatic := 0);
PU600.SetState_Profibus();

PU690(bSetStatusOnAutomatic := bSetStatusOn_PU690,
	bAlgorithmPermission := bAlgorithmPermission);
PU690.SetState_BO();

//valves
SV235.GetState_BI();
SV235(bSetStatusOnAutomatic := bSetStatusOn_SV235,
	bAlgorithmPermission := bAlgorithmPermission);
SV235.SetState_BO();

SV605.GetState_BI();
SV605(bSetStatusOnAutomatic := TRUE,
	bAlgorithmPermission := bAlgorithmPermission);
SV605.SetState_BO();

//RV600 uses heating mode to control inlet temperature into PWT6 (with temperature difference of 7 K of primary and secondary side)
RV600.GetState_AI();
RV600(bSetStatusOnAutomatic := bSetStatusOn_RV600,
	fSetPointAutomatic := fSetPoint,
	bAlgorithmPermission := bAlgorithmPermission,
	fTemperatureExternal := PU235.fTemperatureExternal,
	fThermalPowerExternal := WMZ235.fHeatFlowRate,
	nControlModeAutomatic := 2);
RV600.SetState_AO();

RV640.GetState_AI();
RV640(bSetStatusOnAutomatic := bSetStatusOn_RV640,
	fSetPointAutomatic := fSetPoint_RV640,
	bAlgorithmPermission := bAlgorithmPermission,
	nControlModeAutomatic := 0);
RV640.SetState_AO();

RV660.GetState_AI();
RV660(bSetStatusOnAutomatic := bSetStatusOn_RV660,
	fSetPointAutomatic := fSetPoint_RV660,
	bAlgorithmPermission := bAlgorithmPermission,
	nControlModeAutomatic := 0);
RV660.SetState_AO();

//insert heat counter telegramm from other task
WMZ235(aHeatCounterTelegramm := aTelegramm_WMZ235);

PS600();
PS600.GetState_AI();

TS640();
TS640.GetState_AI();
TS660();
TS660.GetState_AI();

METHOD PROTECTED  CheckError : BOOL
VAR_INPUT
END_VAR
VAR_OUTPUT
	bError : BOOL;
END_VAR
VAR
	bError_PU235 : BOOL;
	bError_PU600 : BOOL;
	bError_SV235 : BOOL;
END_VAR
//check pumps for errors
bError_PU235 := PU235.bError;
bError_PU600 := PU600.bError;

//check valve SV235 for an error
IF SV235.bStatusOn AND PU235.bStatusOn THEN
	bError_SV235 := TRUE;
END_IF

bError := bError_PU235 OR bError_PU600 OR bError_SV235;
END_METHOD

METHOD LocalControl : BOOL
VAR_INPUT
END_VAR
//check for rain
IF NOT stAmbientState.bRain THEN
	bSetStatusOn_PU690 := TRUE;
ELSE
	bSetStatusOn_PU690 := FALSE;
END_IF

//check for time
IF Clock.stClockState.fHour < 12 THEN
	//use west facade	
	fSetPoint_RV660 := 100;
	fSetPoint_RV640 := 0;
ELSE
	//use east facade
	fSetPoint_RV660 := 0;
	fSetPoint_RV640 := 100;
END_IF
END_METHOD

METHOD PROTECTED  Operational : BOOL
VAR_INPUT
END_VAR
VAR_OUTPUT
	bSwitchToWorking : BOOL := FALSE;
END_VAR
bSetStatusOn_PU235 := TRUE;
bSetStatusOn_PU600 := TRUE;
LocalControl();

IF PU235.bStatusOn AND PU600.bStatusOn THEN
	bSwitchToWorking := TRUE;
END_IF;
END_METHOD

METHOD PROTECTED  RampDown : BOOL
VAR_INPUT
END_VAR
VAR_OUTPUT
	bRampDownFinished : BOOL := FALSE;
END_VAR
bSetStatusOn_PU600 := FALSE;
bSetStatusOn_PU235 := FALSE;
bSetStatusOn_PU690 := FALSE;
bSetStatusOn_SV235 := FALSE;
bSetStatusOn_RV600 := FALSE;
bSetStatusOn_RV640 := FALSE;
bSetStatusOn_RV660 := FALSE;
bStartTimer := TRUE;

IF Timer.Q THEN
	bRampDownFinished := TRUE;
	bStartTimer := FALSE;
END_IF
END_METHOD

METHOD PROTECTED  RampUp : BOOL
VAR_INPUT
END_VAR
VAR_OUTPUT
	bRampUpFinished : BOOL := FALSE;
END_VAR
bSetStatusOn_SV235 := TRUE;
bSetStatusOn_RV600 := TRUE;
bSetStatusOn_RV640 := TRUE;
bSetStatusOn_RV660 := TRUE;
bStartTimer := TRUE;

IF Timer.Q THEN
	bRampUpFinished := TRUE;
	bStartTimer := FALSE; //resets timer
END_IF

//check for rain
LocalControl();
END_METHOD

METHOD PROTECTED   SetSetPointLimits : BOOL
VAR_INPUT
END_VAR
aSetPointLimits[1] := localDefaultParameters.aSetPointLimitsTemperature[1];
aSetPointLimits[2] := localDefaultParameters.aSetPointLimitsTemperature[2];
END_METHOD

METHOD PROTECTED  SetState : BOOL
VAR_INPUT
END_VAR
VAR_OUTPUT
END_VAR
fOperatingPoint := PU235.fTemperatureExternal;

controlState.bStatusOn := bSetStatusOn;
setPointState.aSetPointLimits := aSetPointLimits;
setPointState.fSetPoint := fSetPoint;
setPointState.fOperatingPoint := fOperatingPoint;
setPointState.sSetPointUnit := 'degreeC';
setPointState.sOperatingPointUnit := 'degreeC';
END_METHOD

METHOD PROTECTED  Working : BOOL
VAR_INPUT
END_VAR
VAR_OUTPUT
	bSwitchToOperational : BOOL := FALSE;
END_VAR
LocalControl();
END_METHOD

END_FUNCTION_BLOCK

// ---- POUs/04 Systems/ConsumerSystems/HNLT/FB_CompressorSystem.TcPOU
FUNCTION_BLOCK FB_CompressorSystem EXTENDS FB_SystemContinous
VAR_INPUT
END_VAR
VAR_OUTPUT
END_VAR
VAR
	//default parameters
	localDefaultParameters : ST_CompressorDefaultParameters;	

	//pumps
	stPU251DefaultParameters : ST_PumpGrundfosMagna3DefaultParameters := (bPumpBeforeApplication := FALSE, tTaskCycleTime := GlobalVariables.tTaskCycleTime_MAIN, tCtrlCycleTime := GlobalVariables.tCtrlCycleTime_MAIN);
	PU251 : FB_PumpGrundfosMagna3 := (ST_DefaultParameters := stPU251DefaultParameters);;

	//valves
	stRV251DefaultParameters : ST_MixingValveDefaultParameters := (bFeedbackSignal := TRUE, tTaskCycleTime := GlobalVariables.tTaskCycleTime_MAIN, tCtrlCycleTime := GlobalVariables.tCtrlCycleTime_MAIN, fOffsetTerminal := 7970);		
	RV251 : FB_MixingValve := (ST_DefaultParameters := stRV251DefaultParameters);
	WMZ251 : FB_MollineC3HeatCounter();
		
	//internal variables
	bSetStatusOn_PU251 : BOOL;
	bSetStatusOn_RV251 : BOOL;
	
	//compressed air valves
	stSVAir1DefaultParameters : ST_DiscreteValveDefaultParameters := (nFeedback := 0);
	stSVAir2DefaultParameters : ST_DiscreteValveDefaultParameters := (nFeedback := 0);
	stSVAir3DefaultParameters : ST_DiscreteValveDefaultParameters := (nFeedback := 0);
	stSVAir4DefaultParameters : ST_DiscreteValveDefaultParameters := (nFeedback := 0);
	stSVAir5DefaultParameters : ST_DiscreteValveDefaultParameters := (nFeedback := 0);
	stSVAir6DefaultParameters : ST_DiscreteValveDefaultParameters := (nFeedback := 0);
	SVAir1 : FB_DiscreteValve := (ST_DefaultParameters := stSVAir1DefaultParameters);
	SVAir2 : FB_DiscreteValve := (ST_DefaultParameters := stSVAir2DefaultParameters);
	SVAir3 : FB_DiscreteValve := (ST_DefaultParameters := stSVAir3DefaultParameters);
	SVAir4 : FB_DiscreteValve := (ST_DefaultParameters := stSVAir4DefaultParameters);
	SVAir5 : FB_DiscreteValve := (ST_DefaultParameters := stSVAir5DefaultParameters);
	SVAir6 : FB_DiscreteValve := (ST_DefaultParameters := stSVAir6DefaultParameters);
	
END_VAR

MAIN();

PU251.GetState_Profibus();
PU251(bSetStatusOnAutomatic := bSetStatusOn_PU251,
	bAlgorithmPermission := bAlgorithmPermission,
	fSetPointAutomatic := 70,
	nControlModeAutomatic := 0);
PU251.SetState_Profibus();

//external temperature should be measured with external sensor after putting sensor into supply pipe
RV251.GetState_AI();
RV251(bSetStatusOnAutomatic := bSetStatusOn_RV251,
	fSetPointAutomatic := fSetPoint-5,
	bAlgorithmPermission := bAlgorithmPermission,
	nControlModeAutomatic := 2,
	fThermalPowerExternal := WMZ251.fHeatFlowRate,
	fTemperatureExternal := PU251.fTemperatureInternal);
RV251.SetState_AO();

WMZ251(aHeatCounterTelegramm := Telegramm_WZ_Druckluftkompressor);

SVAir1.GetState_BI();
SVAir1(bSetStatusOnAutomatic := TRUE,
	bAlgorithmPermission := bAlgorithmPermission);
SVAir1.SetState_BO();

SVAir2.GetState_BI();
SVAir2(bSetStatusOnAutomatic := TRUE,
	bAlgorithmPermission := bAlgorithmPermission);
SVAir2.SetState_BO();

SVAir3.GetState_BI();
SVAir3(bSetStatusOnAutomatic := TRUE,
	bAlgorithmPermission := bAlgorithmPermission);
SVAir3.SetState_BO();

SVAir4.GetState_BI();
SVAir4(bSetStatusOnAutomatic := TRUE,
	bAlgorithmPermission := bAlgorithmPermission);
SVAir4.SetState_BO();

SVAir5.GetState_BI();
SVAir5(bSetStatusOnAutomatic := TRUE,
	bAlgorithmPermission := bAlgorithmPermission);
SVAir5.SetState_BO();

SVAir6.GetState_BI();
SVAir6(bSetStatusOnAutomatic := TRUE,
	bAlgorithmPermission := bAlgorithmPermission);
SVAir6.SetState_BO();

METHOD PROTECTED  CheckError : BOOL
VAR_INPUT
END_VAR
VAR_OUTPUT
	bError : BOOL;
END_VAR
bError := PU251.bError;
END_METHOD

METHOD PROTECTED  Operational : BOOL
VAR_INPUT
END_VAR
VAR_OUTPUT
	bSwitchToWorking : BOOL := FALSE;
END_VAR
bSetStatusOn_PU251 := TRUE;

IF PU251.bStatusOn THEN
	bSwitchToWorking := TRUE;
END_IF
END_METHOD

METHOD PROTECTED  RampDown : BOOL
VAR_INPUT
END_VAR
VAR_OUTPUT
	bRampDownFinished : BOOL := FALSE;
END_VAR
bSetStatusOn_PU251 := FALSE;

IF NOT PU251.bStatusOn THEN
	bSetStatusOn_RV251 := FALSE;
END_IF
END_METHOD

METHOD PROTECTED  RampUp : BOOL
VAR_INPUT
END_VAR
VAR_OUTPUT
	bRampUpFinished : BOOL := FALSE;
END_VAR
bSetStatusOn_RV251 := TRUE;
bRampUpFinished := TRUE;
END_METHOD

METHOD PROTECTED   SetSetPointLimits : BOOL
VAR_INPUT
END_VAR
aSetPointLimits[1] := localDefaultParameters.aSetPointLimitsTemperature[1];
aSetPointLimits[2] := localDefaultParameters.aSetPointLimitsTemperature[2];
END_METHOD

METHOD PROTECTED  SetState : BOOL
VAR_INPUT
END_VAR
VAR_OUTPUT
END_VAR
fOperatingPoint := PU251.fTemperatureInternal;

controlState.bStatusOn := bSetStatusOn;
setPointState.aSetPointLimits := aSetPointLimits;
setPointState.fSetPoint := fSetPoint;
setPointState.fOperatingPoint := fOperatingPoint;
setPointState.sSetPointUnit := 'degreeC';
setPointState.sOperatingPointUnit := 'degreeC';
END_METHOD

METHOD PROTECTED  Working : BOOL
VAR_INPUT
END_VAR
VAR_OUTPUT
	bSwitchToOperational : BOOL := FALSE;
END_VAR
//empty method
END_METHOD

END_FUNCTION_BLOCK

// ---- POUs/04 Systems/ConsumerSystems/HNLT/FB_AnnealingOvenSealingSystem.TcPOU
FUNCTION_BLOCK FB_AnnealingOvenSealingSystem EXTENDS FB_SystemContinous
VAR_INPUT
END_VAR
VAR_OUTPUT
END_VAR
VAR
	//default parameters
	localDefaultParameters : ST_AnnealingOvenExhaustGasDefaultParameters;

	//pumps
	stPU261DefaultParameters : ST_PumpGrundfosMagna3DefaultParameters := (bPumpBeforeApplication := FALSE, tTaskCycleTime := GlobalVariables.tTaskCycleTime_MAIN, tCtrlCycleTime := GlobalVariables.tCtrlCycleTime_MAIN);
	PU261 : FB_PumpGrundfosMagna3 := (ST_DefaultParameters := stPU261DefaultParameters);

	//valves
	stRV261DefaultParameters : ST_MixingValveDefaultParameters := (bFeedbackSignal := TRUE, fControllerAmplification := 5, tControllerIntegralTime := T#100S, fOutMinLimit := 50, tTaskCycleTime := GlobalVariables.tCtrlCycleTime_MAIN, tCtrlCycleTime := GlobalVariables.tCtrlCycleTime_MAIN, fOffsetTerminal := 7970);
	RV261 : FB_MixingValve := (ST_DefaultParameters := stRV261DefaultParameters);
	
	//sensors	
	WMZ261 : FB_MollineC3HeatCounter;
	
	//internal variables
	bSetStatusOn_PU261 : BOOL;
	bSetStatusOn_RV261 : BOOL;
END_VAR

MAIN();

//pumps
PU261.GetState_Profibus();
PU261(bSetStatusOnAutomatic := bSetStatusOn_PU261,
	fSetPointAutomatic := 100,
	bAlgorithmPermission := bAlgorithmPermission,
	nControlModeAutomatic := 0);
PU261.SetState_Profibus();

//valves
RV261.GetState_AI();
RV261(bSetStatusOnAutomatic := bSetStatusOn_RV261,
	fSetPointAutomatic := fSetPoint,
	bAlgorithmPermission := bAlgorithmPermission,
	fTemperatureExternal := WMZ261.fReturnTemperature,
	fThermalPowerExternal := WMZ261.fHeatFlowRate,
	nControlModeAutomatic := 2);
RV261.SetState_AO();

WMZ261(aHeatCounterTelegramm := Telegramm_WZ_Ofenkuehlung);

METHOD PROTECTED  CheckError : BOOL
VAR_INPUT
END_VAR
VAR_OUTPUT
	bError : BOOL;
END_VAR
bError := PU261.bError;
END_METHOD

METHOD PROTECTED  Operational : BOOL
VAR_INPUT
END_VAR
VAR_OUTPUT
	bSwitchToWorking : BOOL := FALSE;
END_VAR
bSetStatusOn_PU261 := TRUE;

IF PU261.bStatusOn THEN
	bSwitchToWorking := TRUE;
END_IF
END_METHOD

METHOD PROTECTED  RampDown : BOOL
VAR_INPUT
END_VAR
VAR_OUTPUT
	bRampDownFinished : BOOL := FALSE;
END_VAR
bSetStatusOn_PU261 := FALSE;

IF NOT PU261.bStatusOn THEN
	bSetStatusOn_RV261 := FALSE;
	IF RV261.fOperatingPoint<10 THEN
		bRampDownFinished := TRUE;
	END_IF
END_IF
END_METHOD

METHOD PROTECTED  RampUp : BOOL
VAR_INPUT
END_VAR
VAR_OUTPUT
	bRampUpFinished : BOOL := FALSE;
END_VAR
bSetStatusOn_RV261 := TRUE;
bRampUpFinished := TRUE;
END_METHOD

METHOD PROTECTED   SetSetPointLimits : BOOL
VAR_INPUT
END_VAR
aSetPointLimits[1] := localDefaultParameters.aSetPointLimitsTemperature[1];
aSetPointLimits[2] := localDefaultParameters.aSetPointLimitsTemperature[2];
END_METHOD

METHOD PROTECTED  SetState : BOOL
VAR_INPUT
END_VAR
VAR_OUTPUT
END_VAR
fOperatingPoint := WMZ261.fReturnTemperature;

controlState.bStatusOn := bSetStatusOn;
setPointState.aSetPointLimits := aSetPointLimits;
setPointState.fSetPoint := fSetPoint;
setPointState.fOperatingPoint := fOperatingPoint;
setPointState.sSetPointUnit := 'degreeC';
setPointState.sOperatingPointUnit := 'degreeC';
END_METHOD

METHOD PROTECTED  Working : BOOL
VAR_INPUT
END_VAR
VAR_OUTPUT
	bSwitchToOperational : BOOL := FALSE;
END_VAR
//empty method
END_METHOD

END_FUNCTION_BLOCK

// ---- POUs/04 Systems/ConsumerSystems/HNLT/FB_DCSystem.TcPOU
FUNCTION_BLOCK FB_DCSystem EXTENDS FB_SystemContinous
VAR_INPUT
END_VAR
VAR_OUTPUT
END_VAR
VAR
	//default parameters
	localDefaultParameters : ST_DCSystemDefaultParameters;
	
	//pumps
	stPU245DefaultParameters : ST_PumpGrundfosMagna3DefaultParameters := (bPumpBeforeApplication := FALSE, tTaskCycleTime := GlobalVariables.tTaskCycleTime_MAIN, tCtrlCycleTime := GlobalVariables.tCtrlCycleTime_MAIN);
	PU245 : FB_PumpGrundfosMagna3 := (ST_DefaultParameters := stPU245DefaultParameters);;

	//valves
	stSV245DefaultParameters : ST_DiscreteValveDefaultParameters := (nFeedback := 0);
	SV245 : FB_DiscreteValve := (ST_DefaultParameters := stSV245DefaultParameters);
	
	WMZ245 : FB_MollineEHeatCounter;
	
	//internal variables
	bSetStatusOn_PU245 : BOOL;
	bSetStatusOn_SV245 : BOOL;
	
	//timer
	bStartTimer : BOOL;
	Timer : TON;
END_VAR

MAIN();

//use timer because valve has no feedback signal (75 sec)
Timer(IN := bStartTimer,
	PT := T#75S);

SV245.GetState_BI();
SV245(bSetStatusOnAutomatic := bSetStatusOn_SV245,
	bAlgorithmPermission := bAlgorithmPermission);
SV245.SetState_BO();

//pump controls return temperature
PU245.GetState_Profibus();
PU245(bSetStatusOnAutomatic := bSetStatusOn_PU245,
	bAlgorithmPermission := bAlgorithmPermission,
	fSetPointAutomatic := fSetPoint,
	fThermalPowerExternal := WMZ245.fHeatFlowRate,
	nControlModeAutomatic := 3);
PU245.SetState_Profibus();

WMZ245(aHeatCounterTelegramm := aTelegramm_WMZ245);

METHOD PROTECTED  CheckError : BOOL
VAR_INPUT
END_VAR
VAR_OUTPUT
	bError : BOOL;
END_VAR
IF PU245.bError THEN
	bError := TRUE;
END_IF
END_METHOD

METHOD PROTECTED  Operational : BOOL
VAR_INPUT
END_VAR
VAR_OUTPUT
	bSwitchToWorking : BOOL := FALSE;
END_VAR
bSetStatusOn_PU245 := TRUE;

IF PU245.bStatusOn THEN
	bSwitchToWorking := TRUE;
END_IF
END_METHOD

METHOD PROTECTED  RampDown : BOOL
VAR_INPUT
END_VAR
VAR_OUTPUT
	bRampDownFinished : BOOL := FALSE;
END_VAR
bSetStatusOn_PU245 := FALSE;

IF NOT PU245.bStatusOn THEN
	bSetStatusOn_SV245 := FALSE;
	bStartTimer := TRUE;
	IF Timer.Q THEN
		bStartTimer := FALSE;
		bRampDownFinished := TRUE;
	END_IF
END_IF
END_METHOD

METHOD PROTECTED  RampUp : BOOL
VAR_INPUT
END_VAR
VAR_OUTPUT
	bRampUpFinished : BOOL := FALSE;
END_VAR
bSetStatusOn_SV245 := TRUE;
bStartTimer := TRUE;

IF Timer.Q THEN
	bStartTimer := FALSE;
	bRampUpFinished := TRUE;
END_IF
END_METHOD

METHOD PROTECTED   SetSetPointLimits : BOOL
VAR_INPUT
END_VAR
IF  PU245.nControlModeAutomatic = 3 THEN
	aSetPointLimits[1] := localDefaultParameters.aSetPointLimitsTemperatureDifference[1];
	aSetPointLimits[2] := localDefaultParameters.aSetPointLimitsTemperatureDifference[2];
ELSE
	aSetPointLimits[1] := localDefaultParameters.aSetPointLimitsRelativeSpeed[1];
	aSetPointLimits[2] := localDefaultParameters.aSetPointLimitsRelativeSpeed[2];
END_IF
END_METHOD

METHOD PROTECTED  SetState : BOOL
VAR_INPUT
END_VAR
VAR_OUTPUT
END_VAR
fOperatingPoint := PU245.localState.fTemperatureDifference;

controlState.bStatusOn := bSetStatusOn;
setPointState.aSetPointLimits := aSetPointLimits;
setPointState.fSetPoint := fSetPoint;
setPointState.fOperatingPoint := fOperatingPoint;
setPointState.sSetPointUnit := 'K';
setPointState.sOperatingPointUnit := 'K';
END_METHOD

METHOD PROTECTED  Working : BOOL
VAR_INPUT
END_VAR
VAR_OUTPUT
	bSwitchToOperational : BOOL := FALSE;
END_VAR
//empty method
END_METHOD

END_FUNCTION_BLOCK

// ---- POUs/01 Actuators/ConsumerUnits/FB_AnnealingOven.TcPOU
FUNCTION_BLOCK FB_AnnealingOven
VAR_INPUT
END_VAR
VAR_OUTPUT
	bStatusOn_ExhaustGas : BOOL;
	bStatusOn_Sealing : BOOL;
END_VAR
VAR
	//modbus tcp communication
	ModbusReader : FB_MBReadRegs;
	aModbus : ARRAY  [0..61] OF WORD;
	bReadModbus	: BOOL := FALSE;
	bStartTimer : BOOL;
	Timer : TON;
END_VAR

Timer(IN := bStartTimer,
	PT := T#2S);
	
bStartTimer := TRUE;
IF Timer.Q THEN
	bReadModbus := TRUE;
	bStartTimer := FALSE;	
END_IF

ModbusReader(sIPAddr := GlobalVariables.sIP_Annealing_Oven,
	nTCPPort := 502,
	nUnitID := 255,
	nQuantity := 80,
	nMBAddr := 800,
	cbLength := 122,
	pDestAddr := ADR(aModbus),
	bExecute := bReadModbus,
	tTimeout  := T#20S);
bReadModbus := FALSE;

bStatusOn_ExhaustGas := FALSE;
bStatusOn_Sealing := FALSE;

END_FUNCTION_BLOCK

// ---- POUs/01 Actuators/ConsumerUnits/FB_DC.TcPOU
FUNCTION_BLOCK FB_DC
VAR_INPUT
END_VAR
VAR_OUTPUT
	bStatusOn : BOOL;
	bError_Connection : BOOL;
END_VAR
VAR
	OPC_UA				: FB_OPC_UA_READ;
	stOPC_UA_Server		: ST_OPC_UA_Server;
	sOPC_UA_Server_URL 	: STRING;
	sNamespaceName		: STRING;
	aNodes				: ARRAY[1..1] OF ST_OPC_UANode;
	nNodeCount			: UDINT := 1;
	stIndexRange		: ARRAY [1..nMaxIndexRange] OF ST_UAIndexRange;
	currentNode			: UDINT := 1;
	
	// timer
	bStartTimer : BOOL;
	Timer : TON;
END_VAR

sOPC_UA_Server_URL 	:= GlobalVariables.sIP_DC;
sNamespaceName 		:= 'http://www.boschrexroth.com/IndraLogic';

(*Define Nodes to Read*)
aNodes[1].NodeID.sIdentifier			:= '.bHMU_DCBusCharged';
aNodes[1].NodeID.eIdentifierType		:= eUAIdentifierType_String;
aNodes[1].SizeOfDataType				:= DINT_TO_UDINT(eUAType_Boolean);
aNodes[1].NodeAddInfo.nIndexRangeCount 	:= 0;
aNodes[1].NodeAddInfo.stIndexRange		:= stIndexRange;
aNodes[1].TargetVar						:= ADR(bStatusOn);
bError_Connection := OPC_UA.bError_Connection;
Timer(IN := bStartTimer,
	PT := T#5S);

bStartTimer := TRUE;
IF Timer.Q THEN
	OPC_UA(
		stNode				:= aNodes[currentNode],
		sOPC_UA_Server_Url 	:= sOPC_UA_Server_URL,
		sNamespaceName		:= sNamespaceName);
	currentNode := currentNode + 1;
	IF currentNode > nNodeCount THEN
		currentNode := 1;
	END_IF
	bStartTimer := FALSE;
END_IF

END_FUNCTION_BLOCK

// ---- POUs/05 Thermal Networks/FB_HnhtHnltLinkage.TcPOU
FUNCTION_BLOCK FB_HnhtHnltLinkage
VAR_INPUT
	//control struct for hnht hnlt linkage
	controlAutomatic : ST_HnhtHnltLinkageControl;
END_VAR
VAR_OUTPUT
END_VAR
VAR
	HeatExchanger1System : FB_HeatExchanger1System;
	HeatPumpSystem : FB_HeatPumpSystem_HNHT;
	
	
	//internal variables
	bAlgorithmPermission : BOOL;
END_VAR

bAlgorithmPermission := controlAutomatic.bAlgorithmPermission_HNHT AND controlAutomatic.bAlgorithmPermission_HNLT;

HeatExchanger1System(bSetStatusOnAutomatic := controlAutomatic.bSetStatusOn_HeatExchanger1,
	bAlgorithmPermission := bAlgorithmPermission,
	fSetPointAutomatic := controlAutomatic.fFeedTemperature_HNLT_Heating);
	
HeatPumpSystem(bSetStatusOnAutomatic := controlAutomatic.bSetStatusOn_HeatPump,
	bAlgorithmPermission := bAlgorithmPermission,
	fSetPointAutomatic := controlAutomatic.fFeedTemperature_HNHT);

END_FUNCTION_BLOCK

// ---- POUs/04 Systems/LinkageSystems/FB_HeatExchanger1System.TcPOU
FUNCTION_BLOCK FB_HeatExchanger1System EXTENDS FB_SystemContinous
VAR_INPUT
END_VAR
VAR_OUTPUT
END_VAR
VAR
	//default parameters
	localDefaultParameters : ST_HeatExchanger1DefaultParameters;

	//pumps
	stPU315DefaultParameters : ST_PumpGrundfosMagna3DefaultParameters := (tTaskCycleTime := GlobalVariables.tTaskCycleTime_MAIN, tCtrlCycleTime := GlobalVariables.tCtrlCycleTime_MAIN);
	stPU215DefaultParameters : ST_PumpGrundfosMagna3DefaultParameters := (bPumpBeforeApplication := FALSE, tTaskCycleTime := GlobalVariables.tTaskCycleTime_MAIN, tCtrlCycleTime := GlobalVariables.tCtrlCycleTime_MAIN);
	PU315 : FB_PumpGrundfosMagna3 := (ST_DefaultParameters := stPU315DefaultParameters);
	PU215 : FB_PumpGrundfosMagna3 := (ST_DefaultParameters := stPU215DefaultParameters);

	//valves
	stSV215DefaultParameters : ST_DiscreteValveDefaultParameters := (nFeedback := 0);
	stRV315DefaultParameters : ST_MixingValveDefaultParameters := (bFeedbackSignal := TRUE, fControllerAmplification := 1.5, tControllerIntegralTime := T#400S, fOutMinLimit := 25, tTaskCycleTime := GlobalVariables.tTaskCycleTime_MAIN, tCtrlCycleTime := GlobalVariables.tCtrlCycleTime_MAIN, fOffsetTerminal := 7970);
	
	SV215 : FB_DiscreteValve := (ST_DefaultParameters := stSV215DefaultParameters);
	RV315 : FB_MixingValve := (ST_DefaultParameters := stRV315DefaultParameters);
	
	//sensors
	WMZ215 : FB_MollineC3HeatCounter;
	
	//internal variables
	bSetStatusOn_PU315 : BOOL;
	bSetStatusOn_PU215 : BOOL;
	bSetStatusOn_RV315 : BOOL;
	bSetStatusOn_SV215 : BOOL;
	
	bStartTimer : BOOL;
	Timer : TON;
END_VAR

Timer(IN := bStartTimer,
	PT := T#75S);
MAIN();

//pumps
PU315.GetState_Profibus();
PU315(bSetStatusOnAutomatic := bSetStatusOn_PU315,
	fSetPointAutomatic := 100,
	bAlgorithmPermission := bAlgorithmPermission,
	nControlModeAutomatic := 0);
PU315.SetState_Profibus();

PU215.GetState_Profibus();
PU215(bSetStatusOnAutomatic := bSetStatusOn_PU215,
	fSetPointAutomatic := 100,
	bAlgorithmPermission := bAlgorithmPermission,
	nControlModeAutomatic := 0);
PU215.SetState_Profibus();

//valves
RV315.GetState_AI();
RV315(bSetStatusOnAutomatic := bSetStatusOn_RV315,
	bAlgorithmPermission := bAlgorithmPermission,
	fSetPointAutomatic := fSetPoint,
	fTemperatureExternal := PU215.fTemperatureExternal,
	fThermalPowerExternal := WMZ215.fHeatFlowRate,
	nControlModeAutomatic := 1);
RV315.SetState_AO();

SV215.GetState_BI();
SV215(bSetStatusOnAutomatic := bSetStatusOn_SV215,
	bAlgorithmPermission := bAlgorithmPermission);
SV215.SetState_BO();

WMZ215(aHeatCounterTelegramm := Telegramm_WZ_PWT_1);

METHOD PROTECTED  CheckError : BOOL
VAR_INPUT
END_VAR
VAR_OUTPUT
	bError : BOOL;
END_VAR
bError := PU315.bError;
END_METHOD

METHOD PROTECTED  Operational : BOOL
VAR_INPUT
END_VAR
VAR_OUTPUT
	bSwitchToWorking : BOOL := FALSE;
END_VAR
bSetStatusOn_PU315 := TRUE;
bSetStatusOn_PU215 := TRUE;

IF PU315.bStatusOn AND PU215.bStatusOn THEN
	bSwitchToWorking := TRUE;
END_IF
END_METHOD

METHOD PROTECTED  RampDown : BOOL
VAR_INPUT
END_VAR
VAR_OUTPUT
	bRampDownFinished : BOOL := FALSE;
END_VAR
bSetStatusOn_PU215 := FALSE;
bSetStatusOn_PU315 := FALSE;

IF NOT PU315.bStatusOn AND NOT PU215.bStatusOn THEN
	bSetStatusOn_SV215 := FALSE;
	bSetStatusOn_RV315 := FALSE;
	bStartTimer := TRUE;
	IF Timer.Q THEN
		bRampDownFinished := TRUE;
		bStartTimer := FALSE;
	END_IF
END_IF
END_METHOD

METHOD PROTECTED  RampUp : BOOL
VAR_INPUT
END_VAR
VAR_OUTPUT
	bRampUpFinished : BOOL := FALSE;
END_VAR
bSetStatusOn_RV315 := TRUE;
bSetStatusOn_SV215 := TRUE;

bStartTimer := TRUE;
IF Timer.Q THEN
	bStartTimer := FALSE;
	bRampUpFinished := TRUE;
END_IF
END_METHOD

METHOD PROTECTED   SetSetPointLimits : BOOL
VAR_INPUT
END_VAR
aSetPointLimits[1] := localDefaultParameters.aSetPointLimitsTemperature[1];
aSetPointLimits[2] := localDefaultParameters.aSetPointLimitsTemperature[2];
END_METHOD

METHOD PROTECTED  SetState : BOOL
VAR_INPUT
END_VAR
VAR_OUTPUT
END_VAR
fOperatingPoint := PU215.fTemperatureExternal;

controlState.bStatusOn := bSetStatusOn;
setPointState.aSetPointLimits := aSetPointLimits;
setPointState.fSetPoint := fSetPoint;
setPointState.fOperatingPoint := fOperatingPoint;
setPointState.sSetPointUnit := 'degreeC';
setPointState.sOperatingPointUnit := 'degreeC';
END_METHOD

METHOD PROTECTED  Working : BOOL
VAR_INPUT
END_VAR
VAR_OUTPUT
	bSwitchToOperational : BOOL := FALSE;
END_VAR
//empty method
END_METHOD

END_FUNCTION_BLOCK

// ---- POUs/04 Systems/LinkageSystems/FB_HeatPumpSystem_HNHT.TcPOU
FUNCTION_BLOCK FB_HeatPumpSystem_HNHT EXTENDS FB_SystemContinous
VAR_INPUT
END_VAR
VAR_OUTPUT
END_VAR
VAR
	//Vitocal 200-G heat pump
	HeatPump : FB_HeatPump;
	
	//valves
	ST_RV342DefaultParameters : ST_MixingValveDefaultParameters := (fControllerAmplification := 5, tControllerIntegralTime := T#100S, tTaskCycleTime := GlobalVariables.tTaskCycleTime_MAIN, tCtrlCycleTime := GlobalVariables.tCtrlCycleTime_MAIN, fOffsetTerminal := 2900);;
	ST_RV242DefaultParameters : ST_MixingValveDefaultParameters := (fControllerAmplification := 10, tControllerIntegralTime := T#100S, fOutMaxLimit := 100, fOutMinLimit := 35, tTaskCycleTime := GlobalVariables.tTaskCycleTime_MAIN, tCtrlCycleTime := GlobalVariables.tCtrlCycleTime_MAIN, fOffsetTerminal := 3500);
	ST_SV_HNLT_DefaultParameters : ST_DiscreteValveDefaultParameters := (nFeedback := 0);		
	RV342 : FB_MixingValve := (ST_DefaultParameters := ST_RV342DefaultParameters);
	RV242 : FB_MixingValve := (ST_DefaultParameters := ST_RV242DefaultParameters);	
	SV_HNLT : FB_DiscreteValve := (ST_DefaultParameters := ST_SV_HNLT_DefaultParameters);	
	
	//pump
	stPU242DefaultParameters : ST_PumpGrundfosMagna3DefaultParameters := (tTaskCycleTime := GlobalVariables.tTaskCycleTime_MAIN, tCtrlCycleTime := GlobalVariables.tCtrlCycleTime_MAIN, bExternalTemperatureSensor := TRUE);
	PU242 : FB_PumpGrundfosMagna3 := (ST_DefaultParameters := stPU242DefaultParameters);
	
	//internal variables
	bSetStatusOn_HeatPump : BOOL;
	bSetStatusOn_PU242 : BOOL;
	bSetStatusOn_RV342 : BOOL;
	bSetStatusOn_RV242 : BOOL;
	bSetStatusOn_SV_HNLT : BOOL;
	fTemperatureSetPoint_RV242 : REAL;
	
	// timer for SV441, SV442
	bStartTimer_SV : BOOL;
	Timer_SV : TON;
	
	// timer for heat pump
	bStartTimer_HeatPump : BOOL;
	Timer_HeatPump : TON;
	
	//error variable for temperature TS242
	Controller_TS242_Error : FB_CTRL_2POINT;
	Controller_TS242_Error_Parameters : ST_CTRL_2POINT_PARAMS;

	//sensors
	TS242 : FB_TemperatureSensor; //inlet temperature evaporator
	WMZ342 : FB_MollineEHeatCounter;
	EM342 : FB_EmonioP3;
END_VAR

MAIN();
//use timer for cool down during ramp up
Timer_SV(IN := bStartTimer_SV,
	PT := T#30S);
Timer_HeatPump(IN := bStartTimer_HeatPump,
	PT := T#120S);

//valves
SV_HNLT.GetState_BI();
SV_HNLT(bSetStatusOnAutomatic := bSetStatusOn_SV_HNLT,
		bAlgorithmPermission := bAlgorithmPermission);
SV_HNLT.SetState_BO();

//heat pump, use static feed temperature of 64 °C (convertes to max feed temp 65°C in heat pump)
HeatPump.GetState();
HeatPump(bSetStatusOnAutomatic := bSetStatusOn_HeatPump,
	bAlgorithmPermission := bAlgorithmPermission,
	fSetPointAutomatic := 64);
HeatPump.SetState();

//pump
PU242.GetState_Profibus();
PU242(bSetStatusOnAutomatic := bSetStatusOn_PU242,
	fSetPointAutomatic := 50,
	bAlgorithmPermission := bAlgorithmPermission,
	nControlModeAutomatic := 0);
PU242.SetState_Profibus();

//valves
RV242.GetState_AI();
RV242(bSetStatusOnAutomatic := bSetStatusOn_RV242,
	bAlgorithmPermission := bAlgorithmPermission,
	fSetPointAutomatic := fTemperatureSetPoint_RV242,
	fTemperatureExternal := TS242.fTemperature,
	nControlModeAutomatic := 1);
RV242.SetState_AO();

RV342.GetState_AI();
RV342(bSetStatusOnAutomatic := bSetStatusOn_RV342,
	bAlgorithmPermission := bAlgorithmPermission,
	fSetPointAutomatic := 100,
	fThermalPowerExternal := WMZ342.fHeatFlowRate,
	nControlModeAutomatic := 0);
RV342.SetState_AO();

//sensors
WMZ342(aHeatCounterTelegramm := aTelegramm_WMZ342);
TS242();
TS242.GetState_AI();
EM342(sIPAddr := GlobalVariables.sIP_Emonio_HNHT_HeatPump);

METHOD PROTECTED  CheckError : BOOL
VAR_INPUT
END_VAR
VAR_OUTPUT
	bError : BOOL;
END_VAR
Controller_TS242_Error_Parameters.fHysteresisRange := 1;
Controller_TS242_Error_Parameters.tCtrlCycleTime := GlobalVariables.tCtrlCycleTime_MAIN;
Controller_TS242_Error_Parameters.tTaskCycleTime := GlobalVariables.tTaskCycleTime_MAIN;

Controller_TS242_Error(fSetpointValue := 5,
	fActualValue := TS242.fTemperature,
	eMode := eCTRL_MODE_ACTIVE,
	stParams := Controller_TS242_Error_Parameters);

bError := HeatPump.bError OR PU242.bError OR Controller_TS242_Error.bOut;
END_METHOD

METHOD PROTECTED  Operational : BOOL
VAR_INPUT
END_VAR
VAR_OUTPUT
	bSwitchToWorking : BOOL := FALSE;
END_VAR
bSetStatusOn_PU242 := TRUE;

IF PU242.bStatusOn THEN
	bStartTimer_SV := TRUE;
	fTemperatureSetPoint_RV242 := 100;// open RV242 for cooling
	IF Timer_SV.Q THEN
		bStartTimer_SV := FALSE; //resets timer	
		bSetStatusOn_HeatPump := TRUE;
		IF TS242.fTemperature < 15 THEN
			bSwitchToWorking := TRUE;
		END_IF
	END_IF;
END_IF;
END_METHOD

METHOD PROTECTED  RampDown : BOOL
VAR_INPUT
END_VAR
VAR_OUTPUT
	bRampDownFinished : BOOL := FALSE;
END_VAR
bSetStatusOn_HeatPump := FALSE;

bStartTimer_HeatPump := TRUE;

bSetStatusOn_RV342 := FALSE; //close RV342 so heatpump stops
IF Timer_HeatPump.Q THEN	
	bSetStatusOn_RV242 := FALSE; //close RV242
	bStartTimer_SV := TRUE; //wait until RV242 closed
	IF Timer_SV.Q THEN
		bStartTimer_SV := FALSE; //reset sv timer
		bSetStatusOn_PU242 := FALSE; //stop pump
		bSetStatusOn_SV_HNLT := FALSE; //close SV
		IF RV242.fOperatingPoint<10 AND RV342.fOperatingPoint<10 THEN
			bRampDownFinished := TRUE;
		END_IF;
		bStartTimer_HeatPump := FALSE; //reset heatpump timer
	END_IF;
END_IF;
END_METHOD

METHOD PROTECTED  RampUp : BOOL
VAR_INPUT
END_VAR
VAR_OUTPUT
	bRampUpFinished : BOOL := FALSE;
END_VAR
bSetStatusOn_RV242 := TRUE;
bSetStatusOn_RV342 := TRUE;
fTemperatureSetPoint_RV242 := 100;
bSetStatusOn_SV_HNLT := FALSE; //connects CN to heat pump
IF RV342.fOperatingPoint>80 THEN
	bRampUpFinished := TRUE;
END_IF
END_METHOD

METHOD PROTECTED   SetSetPointLimits : BOOL
VAR_INPUT
END_VAR
//heat pump has no continous setpoint (limits are not used) but must be implemented because of abstract method
aSetPointLimits[1] := 10;
aSetPointLimits[2] := 100;
END_METHOD

METHOD PROTECTED  SetState : BOOL
VAR_INPUT
END_VAR
VAR_OUTPUT
END_VAR
fOperatingPoint := WMZ342.fFeedTemperature;

controlState.bStatusOn := HeatPump.bStatusOn;
setPointState.aSetPointLimits := aSetPointLimits;
setPointState.fSetPoint := fSetPoint;
setPointState.fOperatingPoint := fOperatingPoint;
setPointState.sSetPointUnit := 'degreeC';
setPointState.sOperatingPointUnit := 'degreeC';
END_METHOD

METHOD PROTECTED  Working : BOOL
VAR_INPUT
END_VAR
VAR_OUTPUT
	bSwitchToOperational : BOOL := FALSE;
END_VAR
bSetStatusOn_SV_HNLT := TRUE; //connects HNLT to heat pump
fTemperatureSetPoint_RV242 := 20;// temperature setpoint for heating
END_METHOD

END_FUNCTION_BLOCK

// ---- POUs/05 Thermal Networks/FB_HeatingNetworkHighTemperature.TcPOU
FUNCTION_BLOCK FB_HeatingNetworkHighTemperature
VAR_INPUT
	//control struct for hnht
	controlAutomatic : ST_HeatingNetworkHighTemperatureControl;	
	stAmbientState : ST_AmbientState;
END_VAR
VAR_OUTPUT
	{attribute 'OPC.UA.DA' := '1'}
	localState : ST_ThermalNetworkState;
END_VAR
VAR
	//systems
	BufferStorage : FB_BufferStorage;
	CHP1System : FB_CHPSystem;
	CHP2System : FB_CHPSystem;
	CondensingBoilerSystem : FB_CondensingBoilerSystem;
	StaticHeatingSystem : FB_StaticHeatingSystem;
	CentralMachineHeatingSystem : FB_HNHT_CentralMachineHeating;
	AnnealingOvenExhaustGasSystem : FB_AnnealingOvenExhaustGasSystem;
	VSIStorageSystem : FB_VSIStorageSystem;
	
	stSV_SupplyAirDefaultParameters : ST_DiscreteValveDefaultParameters := (nFeedback := 0);
	SV_SupplyAir : FB_DiscreteValve := (ST_DefaultParameters := stSV_SupplyAirDefaultParameters);
		
	//machines
	MAFAC_Java : FB_MAFAC_Java;
	BvL_CleaningSystem : FB_BvL_CleaningSystem;
	AnnealingOvenExhaustGas : FB_AnnealingOven;
	
	//internal variables
	bSetStatusOn_CentralMachineHeating : BOOL;
	bSetStatusOn_AnnealingOven : BOOL;
END_VAR

//buffer storage system
BufferStorage();
localState.fUpperTemperature := BufferStorage.localState.fUpperTemperature;
localState.fMidTemperature := BufferStorage.localState.fMidTemperature;
localState.fLowerTemperature := BufferStorage.localState.fLowerTemperature;
localState.fUpperTemperature_ActiveStorage := VSIStorageSystem.localStorageState.fUpperTemperature;
localState.fLowerTemperature_ActiveStorage := VSIStorageSystem.localStorageState.fLowerTemperature;

//producer
CHP1System(bSetStatusOnAutomatic := controlAutomatic.bSetStatusOn_CHP1,
	bAlgorithmPermission := controlAutomatic.bAlgorithmPermission,
	fSetPointAutomatic := controlAutomatic.fFeedTemperature,
	aHeatCounterTelegramm := Telegramm_WZ_BHKW_1,
	aElectricityMeterTelegramm := Telegramm_SZ_BHKW_321,
	aGasMeterTelegramm := Telegramm_GZ_BHKW_321,
	sIPAddressCHP := GlobalVariables.sIP_CHP1);

CHP2System(bSetStatusOnAutomatic := controlAutomatic.bSetStatusOn_CHP2,
	bAlgorithmPermission := controlAutomatic.bAlgorithmPermission,
	fSetPointAutomatic := controlAutomatic.fFeedTemperature,
	aHeatCounterTelegramm := Telegramm_WZ_BHKW_2,
	aElectricityMeterTelegramm := Telegramm_SZ_BHKW_322,
	aGasMeterTelegramm := Telegramm_GZ_BHKW_322,
	sIPAddressCHP := GlobalVariables.sIP_CHP2);

SV_SupplyAir.GetState_BI();
SV_SupplyAir(bSetStatusOnAutomatic := CHP1System.bSetStatusOnFeedback OR CHP2System.bSetStatusOnFeedback,
	bAlgorithmPermission := controlAutomatic.bAlgorithmPermission);
SV_SupplyAir.SetState_BO();

CondensingBoilerSystem(bSetStatusOnAutomatic := controlAutomatic.bSetStatusOn_CondensingBoiler,
	bAlgorithmPermission := controlAutomatic.bAlgorithmPermission,
	fSetPointAutomatic := controlAutomatic.fFeedTemperature);
				
//consumer
StaticHeatingSystem(bSetStatusOnAutomatic := controlAutomatic.bSetStatusOn_StaticHeating,
	bAlgorithmPermission := controlAutomatic.bAlgorithmPermission,
	fSetPointAutomatic := 0,
	stAmbientState := stAmbientState);
	
MAFAC_Java();
BvL_CleaningSystem();
bSetStatusOn_CentralMachineHeating := BvL_CleaningSystem.bHNHT_Demand;

CentralMachineHeatingSystem(bSetStatusOnAutomatic := bSetStatusOn_CentralMachineHeating,
	bAlgorithmPermission := controlAutomatic.bAlgorithmPermission,
	fSetPointAutomatic := 5); // temperature difference control
	
AnnealingOvenExhaustGas();
bSetStatusOn_AnnealingOven := AnnealingOvenExhaustGas.bStatusOn_ExhaustGas;
AnnealingOvenExhaustGasSystem(bSetStatusOnAutomatic := bSetStatusOn_AnnealingOven,
	bAlgorithmPermission := controlAutomatic.bAlgorithmPermission,
	fSetPointAutomatic := controlAutomatic.fFeedTemperature);
	
VSIStorageSystem(bSetStatusOnAutomatic := controlAutomatic.bSetStatusOn_VSIStorage,
	bAlgorithmPermission := controlAutomatic.bAlgorithmPermission,
	fSetPointAutomatic := 30,
	fTemperatureBufferStorageSetPoint := controlAutomatic.fTargetTemperature,
	fTemperatureBufferStorage := localState.fMidTemperature,
	bLoadingAutomatic := controlAutomatic.bLoading_VSISystem);

END_FUNCTION_BLOCK

// ---- POUs/04 Systems/HeatingSystems/FB_CHPSystem.TcPOU
FUNCTION_BLOCK FB_CHPSystem EXTENDS FB_SystemContinous
VAR_INPUT
	aHeatCounterTelegramm : ARRAY[1..cMBUS_MaxTelegrams] OF ST_MBus_Data2;
	aElectricityMeterTelegramm : ARRAY[1..cMBUS_MaxTelegrams] OF ST_MBus_Data2;
	aGasMeterTelegramm : ARRAY[1..cMBUS_MaxTelegrams] OF ST_MBus_Data2;
	sIPAddressCHP : STRING(15);
END_VAR
VAR_OUTPUT
	bSetStatusOnFeedback : BOOL; //Feedback if CHP unit should be switched on to be sent to supply air valve
END_VAR
VAR	
	//chp
	CHP : FB_CHP;

	//pump
	stPU32xDefaultParameters : ST_PumpGrundfosMagna3DefaultParameters := (bPumpBeforeApplication := FALSE, tTaskCycleTime := GlobalVariables.tTaskCycleTime_MAIN, tCtrlCycleTime := GlobalVariables.tCtrlCycleTime_MAIN);
	PU32x : FB_PumpGrundfosMagna3 := (ST_DefaultParameters := stPU32xDefaultParameters);
	
	//valves
	stSV32xDefaultParameters : ST_DiscreteValveDefaultParameters := (nFeedback := 3);
	stRV32xDefaultParameters : ST_MixingValveDefaultParameters := (bFeedbackSignal := TRUE, fControllerAmplification := 5, tControllerIntegralTime := T#100S, fOutMinLimit := 50,  tTaskCycleTime := GlobalVariables.tTaskCycleTime_MAIN, tCtrlCycleTime := GlobalVariables.tCtrlCycleTime_MAIN, fOffsetTerminal := 7970);	
	SV32x : FB_DiscreteValve := (ST_DefaultParameters := stSV32xDefaultParameters);
	RV32x : FB_MixingValve := (ST_DefaultParameters := stRV32xDefaultParameters);
	
	//sensors
	WMZ32x : FB_MollineC3HeatCounter();
	EM32x : FB_ElectricityMeter_BergDCMI461WP();
	GM32x : FB_GasMeter_Aerius_G4();
	
	PI_Controller				: FB_CTRL_PI;
	PI_Controller_Parameters 	: ST_CTRL_PI_PARAMS;
	
	//internal variables
	bSetStatusOn_CHP   : BOOL;
	bSetStatusOn_PU32x : BOOL;
	bSetStatusOn_SV32x : BOOL;
	bSetStatusOn_RV32x : BOOL;
	
	//timer
	bStartTimer : BOOL;
	Timer : TON;
END_VAR

bSetStatusOnFeedback := bSetStatusOn;

//use timer because valve has no feedback signal (120 sec)
Timer(IN := bStartTimer,
	PT := T#120S);

MAIN();
CHP.GetState();
CHP(fSetPointAutomatic :=  fSetPoint,
	bSetStatusOnAutomatic := bSetStatusOn_CHP,
	bAlgorithmPermission := bAlgorithmPermission,
	nControlModeAutomatic := 1,
	fExternalFeedTemperature := PU32x.fTemperatureInternal,
	sIPAddress := sIPAddressCHP);
CHP.SetState();

SV32x.GetState_BI();
SV32x(bSetStatusOnAutomatic := bSetStatusOn_SV32x,
	bAlgorithmPermission := bAlgorithmPermission);
SV32x.SetState_BO();

RV32x.GetState_AI();
RV32x(fSetPointAutomatic := fSetPoint-20,
	bSetStatusOnAutomatic := bSetStatusOn_RV32x,
	bAlgorithmPermission := bAlgorithmPermission,
	fTemperatureExternal := CHP.fReturnTemperature,
	fThermalPowerExternal := WMZ32x.fHeatFlowRate,
	nControlModeAutomatic := 2);
RV32x.SetState_AO();

PU32x.GetState_Profibus();
PU32x(fSetPointAutomatic := 100,
	bSetStatusOnAutomatic := bSetStatusOn_PU32x,
	bAlgorithmPermission := bAlgorithmPermission,
	nControlModeAutomatic := 0);
PU32x.SetState_Profibus();

WMZ32x(aHeatCounterTelegramm := aHeatCounterTelegramm);
EM32x(aElectricityMeterTelegramm := aElectricityMeterTelegramm);
GM32x(aGasmeterTelegramm := aGasMeterTelegramm);

METHOD PROTECTED  CheckError : BOOL
VAR_INPUT
END_VAR
VAR
	bError_PU32x : BOOL;
	//bError_CHP : BOOL;
END_VAR
VAR_OUTPUT
	bError : BOOL;
END_VAR
//check pumps for errors
bError_PU32x := PU32x.bError;
//bError_CHP := CHP.bError;

//bError := bError_PU32x OR bError_CHP;
bError := bError_PU32x;
END_METHOD

METHOD PROTECTED  Operational : BOOL
VAR_INPUT
END_VAR
VAR_OUTPUT
	bSwitchToWorking : BOOL := FALSE;
END_VAR
bSetStatusOn_PU32x := TRUE;

IF PU32x.bStatusOn THEN
	bSetStatusOn_CHP := TRUE;
	bStartTimer := TRUE;
	IF TIMER.Q THEN
		bSwitchToWorking := TRUE;
		bStartTimer := FALSE;
	END_IF
END_IF
END_METHOD

METHOD PROTECTED  RampDown : BOOL
VAR_INPUT
END_VAR
VAR_OUTPUT
	bRampDownFinished : BOOL := FALSE;
END_VAR
bSetStatusOn_CHP := FALSE;

bStartTimer := TRUE;
IF Timer.Q THEN
	bSetStatusOn_PU32x := FALSE;
	bStartTimer := FALSE;
END_IF

IF NOT PU32x.bStatusOn THEN
	bSetStatusOn_RV32x := FALSE;
	bSetStatusOn_SV32x := FALSE;

	IF SV32x.localState.nPosition = 2 THEN
		bRampDownFinished := TRUE;
	END_IF
END_IF
END_METHOD

METHOD PROTECTED  RampUp : BOOL
VAR_INPUT
END_VAR
VAR_OUTPUT
	bRampUpFinished : BOOL := FALSE;
END_VAR
bSetStatusOn_SV32x := TRUE;
bSetStatusOn_RV32x := TRUE;

IF SV32x.localState.nPosition = 3 THEN
	bRampUpFinished := TRUE;
END_IF
END_METHOD

METHOD PROTECTED   SetSetPointLimits : BOOL
VAR_INPUT
END_VAR
aSetPointLimits[1] := CHP.ST_DefaultParameters.aSetPointLimitsTemperature[1];
aSetPointLimits[2] := CHP.ST_DefaultParameters.aSetPointLimitsTemperature[2];
END_METHOD

METHOD PROTECTED  SetState : BOOL
VAR_INPUT
END_VAR
VAR_OUTPUT
END_VAR
fOperatingPoint := PU32x.fTemperatureInternal;

controlState.bStatusOn := bSetStatusOn;
setPointState.aSetPointLimits := aSetPointLimits;
setPointState.fSetPoint := fSetPoint;
setPointState.fOperatingPoint := fOperatingPoint;
setPointState.sSetPointUnit := 'degreeC';
setPointState.sOperatingPointUnit := 'degreeC';
END_METHOD

METHOD PROTECTED  Working : BOOL
VAR_INPUT
END_VAR
VAR_OUTPUT
	bSwitchToOperational : BOOL := FALSE;
END_VAR
//empty method
END_METHOD

END_FUNCTION_BLOCK

// ---- POUs/01 Actuators/HeatingUnits/FB_CHP.TcPOU
FUNCTION_BLOCK FB_CHP EXTENDS FB_ActuatorContinous
VAR_INPUT
	nControlModeAutomatic : E_CHPControlMode; //control mode: 0 = constant power, 1 = feed temperature
	fExternalFeedTemperature : REAL; //external measurement of feed temperature
	sIPAddress : STRING(15);
END_VAR
VAR_OUTPUT
	fReturnTemperature : REAL;
	bError : BOOL;
END_VAR
VAR
	{attribute 'OPC.UA.DA' := '1'}
	localState : ST_CHPState;
	{attribute 'OPC.UA.DA' := '1'}
	localSetParameters : ST_CHPSetParameters;
	
	//default parameters
	localDefaultParameters : ST_CHPDefaultParameters:= (tTaskCycleTime := GlobalVariables.tTaskCycleTime_MAIN, tCtrlCycleTime := GlobalVariables.tCtrlCycleTime_MAIN);	
	
	//modbus tcp communication
	ModbusReader : FB_MBReadRegs;
	aModbus : ARRAY  [0..61] OF WORD;
	
	//analog converters
	OutputConverter : FB_AnalogOutput(fUpperLimit := 100, fLowerLimit := 0);
	
	//I/O Links
	nSetPoint_OUT			AT %Q* : INT; //Set position linked to terminal
	bSetStatusOn_OUT 		AT %Q* : BOOL; //SetStatus linked to terminal
	bError_IN 				AT %I* : BOOL; //Error state linked to terminal
	
	//modbus
	bReadModbus	: BOOL := FALSE;
	bStartTimer : BOOL;
	Timer : TON;
	
	//internal variables
	nControlMode : E_CHPControlMode;
	fSetPoint_internal 		: REAL;
	
	//controllers
	PI_Controller				: FB_CTRL_PI; 
	PI_Controller_Parameters 	: ST_CTRL_PI_PARAMS;
END_VAR

MAIN();
SelectLocalControlMode();
LocalControl();
OutputConverter(fValue := fSetPoint_internal);
Timer(IN := bStartTimer,
	PT := T#2S);
	
bStartTimer := TRUE;
IF Timer.Q THEN
	bReadModbus := TRUE;
	bStartTimer := FALSE;	
END_IF

ModbusReader(sIPAddr := sIPAddress,
	nTCPPort := 502,
	nUnitID := 255,
	nQuantity := 60,
	nMBAddr := 16384,
	cbLength := 122,
	pDestAddr := ADR(aModbus),
	bExecute := bReadModbus,
	tTimeout  := T#20S);
bReadModbus := FALSE;

fReturnTemperature := localState.fReturnTemperature;

METHOD GetState : BOOL
VAR_INPUT
END_VAR
//local state
CASE WORD_TO_UINT(aModbus[2]) OF
	3:
	controlState.bStatusOn := TRUE;
	
	4:
	localState.bError := TRUE;
ELSE
	controlState.bStatusOn := FALSE;
	localState.bError := FALSE;
END_CASE
bStatusOn := controlState.bStatusOn;
bError := localState.bError;
localState.fCosPhi := WORD_TO_INT(aModbus[59])/1000;
localState.fElectricalPower := WORD_TO_INT(aModbus[52])/10;
localState.fFeedTemperature := WORD_TO_INT(aModbus[26])/10;
localState.fGeneratorCurrent := WORD_TO_INT(aModbus[51])/10;
localState.fGeneratorVoltage := WORD_TO_INT(aModbus[50]);
localState.fGridVoltage := WORD_TO_INT(aModbus[49]);
localState.fOperatingTime := WORD_TO_UINT(aModbus[13]);
localState.fReturnTemperature := WORD_TO_INT(aModbus[25])/10;
localState.fRotationalSpeed := WORD_TO_UINT(aModbus[37]);
localState.fTemperatureCoolingWater := WORD_TO_INT(aModbus[24])/10;
localState.fTemperatureExhaustGas := WORD_TO_INT(aModbus[20]);
localState.nNumberOfStarts := WORD_TO_UINT(aModbus[15]);
localState.nOperationStatus := WORD_TO_UINT(aModbus[2]);

//setpoint state
CASE nControlMode OF
	0: //constant power
	setPointState.fOperatingPoint := WORD_TO_INT(aModbus[4]);
	setPointState.sOperatingPointUnit := 'percent';
	
	1: //feed temperature
	setPointState.fOperatingPoint := localState.fFeedTemperature;
	setPointState.sOperatingPointUnit := 'degreeC';
END_CASE
fOperatingPoint := setPointState.fOperatingPoint;
END_METHOD

METHOD LocalControl : BOOL
VAR_INPUT
END_VAR
//set control parameters
PI_Controller_Parameters.fKp 				:= localDefaultParameters.fControllerAmplification;
PI_Controller_Parameters.tTn 				:= localDefaultParameters.tControllerIntegralTime;
PI_Controller_Parameters.fOutMaxLimit		:= 100.0;
PI_Controller_Parameters.fOutMinLimit		:= 0;
PI_Controller_Parameters.tTaskCycleTime		:= localDefaultParameters.tTaskCycleTime;
PI_Controller_Parameters.tCtrlCycleTime		:= localDefaultParameters.tCtrlCycleTime;
PI_Controller_Parameters.bARWOnIPartOnly	:= TRUE;

CASE nControlMode OF
	0: //constant power
	fSetPoint_internal := (fSetPoint - 50.0) * (100.0 / 50.0); //mapping from allowed setpointrange 50-100 to chp range 0-100
	
	1: //feed temperature
	PI_Controller (
			fSetpointValue	:= fSetPoint,
			fActualValue	:= fExternalFeedTemperature,
			fManSyncValue	:= 0,
			bSync			:= FALSE,
			eMode			:= 2, (* mode active *)
			bHold			:= FALSE,
			stParams		:= PI_Controller_Parameters);
	fSetPoint_internal := LREAL_TO_REAL(PI_Controller.fOut);
END_CASE
END_METHOD

METHOD SelectLocalControlMode : BOOL
VAR_INPUT
END_VAR
IF control.bManualModeActivated THEN
	nControlMode := localSetParameters.nControlModeManual;
ELSIF control.bAlgorithmModeActivated AND bAlgorithmPermission THEN
	nControlMode := localSetParameters.nControlModeAlgorithm;
ELSE
	nControlMode := nControlModeAutomatic;
END_IF
END_METHOD

METHOD PROTECTED  SetSetPointLimits : BOOL
VAR_INPUT
END_VAR
CASE nControlMode OF
	0: //constant power
	aSetPointLimits := localDefaultParameters.aSetPointLimitsConstantPower;

	1: //feed temperature
	aSetPointLimits := localDefaultParameters.aSetPointLimitsTemperature;
END_CASE
END_METHOD

METHOD SetState : BOOL
VAR_INPUT
END_VAR
setPointState.fSetPoint := fSetPoint;
setPointState.aSetPointLimits := aSetPointLimits;
CASE nControlMode OF
	0: //constant power
	setPointState.sSetPointUnit := 'percent';
	
	1: //feed temperature
	setPointState.sSetPointUnit := 'degreeC';
END_CASE

nSetPoint_OUT := OutputConverter.nValue;  //converts real setpoint for terminal
bSetStatusOn_OUT := bSetStatusOn;
END_METHOD

PROPERTY ST_DefaultParameters : REFERENCE TO ST_CHPDefaultParameters
GET
ST_DefaultParameters REF= localDefaultParameters;
END_GET
SET
localDefaultParameters := ST_DefaultParameters;
END_SET
END_PROPERTY

END_FUNCTION_BLOCK

// ---- POUs/04 Systems/HeatingSystems/FB_CondensingBoilerSystem.TcPOU
FUNCTION_BLOCK FB_CondensingBoilerSystem EXTENDS FB_SystemContinous
VAR_INPUT
END_VAR
VAR_OUTPUT
END_VAR
VAR
	//default parameters
	localDefaultParameters : ST_CondensingBoilerDefaultParameters;

	//condensing boiler
	CondensingBoiler : FB_CondensingBoiler;
	
	// timer for condensing boiler
	bStartTimer_CondensingBoiler : BOOL;
	Timer_CondensingBoiler : TON;
	
	//valves
	ST_SV331DefaultParameters : ST_DiscreteValveDefaultParameters := (nFeedback := 3);
	ST_RV331DefaultParameters :  ST_MixingValveDefaultParameters := (bFeedbackSignal := TRUE, fControllerAmplification := 1, tControllerIntegralTime := T#100S, fOutMinLimit := 50,  tTaskCycleTime := GlobalVariables.tTaskCycleTime_MAIN, tCtrlCycleTime := GlobalVariables.tCtrlCycleTime_MAIN, fOffsetTerminal := 7970);			
	SV331 : FB_DiscreteValve := (ST_DefaultParameters := ST_SV331DefaultParameters);
	RV331 : FB_MixingValve := (ST_DefaultParameters := ST_RV331DefaultParameters);	
	
	//heat counters
	WMZ331 : FB_MollineC3HeatCounter;
	GM331 : FB_EmonioP3;
	
	//internal variables
	bSetStatusOn_CondensingBoiler : BOOL;
	bSetStatusOn_SV331 : BOOL;
	bStatusOn_SV331 : BOOL;
	bSetStatusOn_RV331 : BOOL;
	bStatusOn_RV331 : BOOL;
END_VAR

MAIN();

Timer_CondensingBoiler(IN := bStartTimer_CondensingBoiler,
	PT := T#120S);

CondensingBoiler.GetState();
CondensingBoiler(bSetStatusOnAutomatic := bSetStatusOn_CondensingBoiler,
	bAlgorithmPermission := bAlgorithmPermission,
	fSetPointAutomatic := fSetPoint);
CondensingBoiler.SetState();

SV331.GetState_BI();
SV331(bSetStatusOnAutomatic := bSetStatusOn_SV331,
	bAlgorithmPermission := bAlgorithmPermission);
SV331.SetState_BO();

RV331.GetState_AI();
RV331(bSetStatusOnAutomatic := bSetStatusOn_RV331,
	fSetPointAutomatic := 100,
	bAlgorithmPermission := bAlgorithmPermission,
	nControlModeAutomatic := 0,
	fThermalPowerExternal := WMZ331.fHeatFlowRate);
RV331.SetState_AO();

//sensors
WMZ331(aHeatCounterTelegramm := Telegramm_WZ_Brennwerttherme);
GM331(sIPAddr := GlobalVariables.sIP_Emonio_CondensingBoiler);

METHOD PROTECTED  CheckError : BOOL
VAR_INPUT
END_VAR
VAR_OUTPUT
	bError : BOOL;
END_VAR
//empty method because condensing boiler has no feedback signal
END_METHOD

METHOD PROTECTED  Operational : BOOL
VAR_INPUT
END_VAR
VAR_OUTPUT
	bSwitchToWorking : BOOL := FALSE;
END_VAR
bSetStatusOn_CondensingBoiler := TRUE;
bSwitchToWorking := TRUE;
END_METHOD

METHOD PROTECTED  RampDown : BOOL
VAR_INPUT
END_VAR
VAR_OUTPUT
	bRampDownFinished : BOOL := FALSE;
END_VAR
bSetStatusOn_CondensingBoiler := FALSE;
bStartTimer_CondensingBoiler := TRUE;

IF Timer_CondensingBoiler.Q THEN
	bSetStatusOn_SV331 := FALSE;
	bSetStatusOn_RV331 := FALSE;
	bStartTimer_CondensingBoiler := FALSE;
	bRampDownFinished := TRUE;
END_IF
END_METHOD

METHOD PROTECTED  RampUp : BOOL
VAR_INPUT
END_VAR
VAR_OUTPUT
	bRampUpFinished : BOOL := FALSE;
END_VAR
bSetStatusOn_SV331 := TRUE;
bSetStatusOn_RV331 := TRUE;
bStartTimer_CondensingBoiler := TRUE;

IF Timer_CondensingBoiler.Q THEN
	bStartTimer_CondensingBoiler := TRUE;
	bStartTimer_CondensingBoiler := FALSE;
	bRampUpFinished := TRUE;
END_IF
END_METHOD

METHOD PROTECTED   SetSetPointLimits : BOOL
VAR_INPUT
END_VAR
aSetPointLimits[1] := localDefaultParameters.aSetPointLimitsTemperature[1];
aSetPointLimits[2] := localDefaultParameters.aSetPointLimitsTemperature[2];
END_METHOD

METHOD PROTECTED  SetState : BOOL
VAR_INPUT
END_VAR
VAR_OUTPUT
END_VAR
fOperatingPoint := WMZ331.fFeedTemperature;

controlState.bStatusOn := bSetStatusOn;
setPointState.aSetPointLimits := aSetPointLimits;
setPointState.fSetPoint := fSetPoint;
setPointState.fOperatingPoint := fOperatingPoint;
setPointState.sSetPointUnit := 'degreeC';
setPointState.sOperatingPointUnit := 'degreeC';
END_METHOD

METHOD PROTECTED  Working : BOOL
VAR_INPUT
END_VAR
VAR_OUTPUT
	bSwitchToOperational : BOOL := FALSE;
END_VAR
//empty method
END_METHOD

END_FUNCTION_BLOCK

// ---- POUs/01 Actuators/HeatingUnits/FB_CondensingBoiler.TcPOU
FUNCTION_BLOCK FB_CondensingBoiler EXTENDS FB_ActuatorContinous
VAR_INPUT
END_VAR
VAR_OUTPUT
	bError : BOOL;
END_VAR
VAR
	{attribute 'OPC.UA.DA' := '1'}
	localState : ST_CondensingBoilerState;
	
	//default parameters
	localDefaultParameters : ST_CondensingBoilerDefaultParameters;
	
	//analog converters
	OutputConverter : FB_AnalogOutput(fUpperLimit := 100, fLowerLimit := 0);
	
	//I/O Links
	nSetPoint_OUT			AT %Q* : INT;
	bSetStatusOn_OUT 		AT %Q* : BOOL;
	bStatusOn_IN			AT %I* : BOOL;
	bError_IN 				AT %I* : BOOL;
END_VAR

MAIN();
OutputConverter(fValue := fSetPoint);

METHOD GetState : BOOL
VAR_INPUT
END_VAR
//local state
controlState.bStatusOn := bStatusOn_IN;
localState.bError := bError_IN;
bStatusOn := controlState.bStatusOn;
bError := localState.bError;
END_METHOD

METHOD PROTECTED  SetSetPointLimits : BOOL
VAR_INPUT
END_VAR
aSetPointLimits[1] := localDefaultParameters.aSetPointLimitsTemperature[1];
aSetPointLimits[2] := localDefaultParameters.aSetPointLimitsTemperature[2];
END_METHOD

METHOD SetState : BOOL
VAR_INPUT
END_VAR
setPointState.fSetPoint := fSetPoint;
setPointState.aSetPointLimits := aSetPointLimits;
setPointState.sSetPointUnit := 'degreeC';

nSetPoint_OUT := OutputConverter.nValue;  //converts real setpoint for terminal
bSetStatusOn_OUT := bSetStatusOn;
END_METHOD

PROPERTY ST_DefaultParameters : REFERENCE TO ST_CondensingBoilerDefaultParameters
GET
ST_DefaultParameters REF= localDefaultParameters;
END_GET
SET
localDefaultParameters := ST_DefaultParameters;
END_SET
END_PROPERTY

END_FUNCTION_BLOCK

// ---- POUs/04 Systems/ConsumerSystems/HNHT/FB_StaticHeatingSystem.TcPOU
FUNCTION_BLOCK FB_StaticHeatingSystem EXTENDS FB_SystemContinous
VAR_INPUT
	stAmbientState : ST_AmbientState;
END_VAR
VAR_OUTPUT
END_VAR
VAR
	//default parameters
	localDefaultParameters : ST_StaticHeatingDefaultParameters;	
	
	//pumps
	stPU350DefaultParameters : ST_PumpGrundfosMagna3DefaultParameters;
	PU350 : FB_PumpGrundfosMagna3 := (ST_DefaultParameters := stPU350DefaultParameters);	
	
	//valves
	stRV350DefaultParameters : ST_MixingValveDefaultParameters := (bFeedbackSignal := FALSE, tTaskCycleTime := GlobalVariables.tTaskCycleTime_MAIN, tCtrlCycleTime := GlobalVariables.tCtrlCycleTime_MAIN);	
	RV350 : FB_MixingValve := (ST_DefaultParameters := stRV350DefaultParameters);
	
	//sensors
	WMZ350 : FB_MollineEHeatCounter;
	
	//internal variables
	bSetStatusOn_PU350 		: BOOL;
	bSetStatusOn_RV350 		: BOOL;
	fSetPoint_Internal 		: REAL;	
	
	//characteristic curve
	CharacteristicCurve 			: FB_CTRL_FLOW_TEMP_SETPOINT_GEN;
	CharacteristicCurve_Parameters	: ST_CTRL_FLOW_TEMP_SETPOINT_GEN_PARAMS;
END_VAR

LocalControl();
fSetPointAutomatic := fSetPoint_Internal;
MAIN();

//pumps
PU350.GetState_Profibus();
PU350(bSetStatusOnAutomatic := bSetStatusOn_PU350,
	fSetPointAutomatic := 100,
	bAlgorithmPermission := bAlgorithmPermission,
	fThermalPowerExternal := WMZ350.fHeatFlowRate,
	nControlModeAutomatic := 0);
PU350.SetState_Profibus();

//valves in thermal networks
RV350.GetState_AI();
RV350(bSetStatusOnAutomatic := bSetStatusOn_RV350,
	fSetPointAutomatic := fSetPoint,
	bAlgorithmPermission := bAlgorithmPermission,
	fTemperatureExternal := PU350.fTemperatureInternal,
	fThermalPowerExternal := WMZ350.fHeatFlowRate,
	nControlModeAutomatic := 1);
RV350.SetState_AO();

WMZ350(aHeatCounterTelegramm := aTelegramm_WMZ350);

METHOD PROTECTED  CheckError : BOOL
VAR_INPUT
END_VAR
VAR_OUTPUT
	bError : BOOL;
END_VAR
VAR
END_VAR
bError :=  PU350.bError;
END_METHOD

METHOD PRIVATE LocalControl : BOOL
VAR_INPUT
END_VAR
VAR
END_VAR
CharacteristicCurve_Parameters.fAmbientTempMax := localDefaultParameters.aLimitsAmbientTemperature[2];
CharacteristicCurve_Parameters.fAmbientTempMin := localDefaultParameters.aLimitsAmbientTemperature[1];
CharacteristicCurve_Parameters.fForeRunTempMax := localDefaultParameters.aLimitsFeedTemperature[1];
CharacteristicCurve_Parameters.fForeRunTempMin := localDefaultParameters.aLimitsFeedTemperature[2];
CharacteristicCurve_Parameters.tCtrlCycleTime := GlobalVariables.tCtrlCycleTime_MAIN;
CharacteristicCurve_Parameters.tTaskCycleTime := GlobalVariables.tTaskCycleTime_MAIN;

CharacteristicCurve(fAmbientTemperature := stAmbientState.fOutsideTemperature,
	fOffsetTemperature := 0,
	bLimitFlowTemp := TRUE,
	stParams := CharacteristicCurve_Parameters);
fSetPoint_Internal := LREAL_TO_REAL(CharacteristicCurve.fOut);
END_METHOD

METHOD PROTECTED  Operational : BOOL
VAR_INPUT
END_VAR
VAR_OUTPUT
	bSwitchToWorking : BOOL := FALSE;
END_VAR
bSetStatusOn_PU350 := TRUE;

IF PU350.bStatusOn THEN
	bSwitchToWorking := TRUE;
END_IF
END_METHOD

METHOD PROTECTED  RampDown : BOOL
VAR_INPUT
END_VAR
VAR_OUTPUT
	bRampDownFinished : BOOL := FALSE;
END_VAR
bSetStatusOn_PU350 := FALSE;
bSetStatusOn_RV350 := FALSE;
	
IF NOT PU350.bStatusOn THEN
	bRampDownFinished := TRUE;		
END_IF
END_METHOD

METHOD PROTECTED  RampUp : BOOL
VAR_INPUT
END_VAR
VAR_OUTPUT
	bRampUpFinished : BOOL := FALSE;
END_VAR
bSetStatusOn_RV350 := TRUE;
bRampUpFinished := TRUE;
END_METHOD

METHOD PROTECTED   SetSetPointLimits : BOOL
VAR_INPUT
END_VAR
aSetPointLimits[1] := localDefaultParameters.aSetPointLimitsTemperature[1];
aSetPointLimits[2] := localDefaultParameters.aSetPointLimitsTemperature[2];
END_METHOD

METHOD PROTECTED  SetState : BOOL
VAR_INPUT
END_VAR
VAR_OUTPUT
END_VAR
fOperatingPoint := PU350.fTemperatureInternal;

controlState.bStatusOn := bSetStatusOn;
setPointState.aSetPointLimits := aSetPointLimits;
setPointState.fSetPoint := fSetPoint;
setPointState.fOperatingPoint := fOperatingPoint;
setPointState.sSetPointUnit := 'degreeC';
setPointState.sOperatingPointUnit := 'degreeC';
END_METHOD

METHOD PROTECTED  Working : BOOL
VAR_INPUT
END_VAR
VAR_OUTPUT
	bSwitchToOperational : BOOL := FALSE;
END_VAR
//empty method
END_METHOD

END_FUNCTION_BLOCK

// ---- POUs/04 Systems/ConsumerSystems/HNHT/FB_HNHT_CentralMachineHeating.TcPOU
FUNCTION_BLOCK FB_HNHT_CentralMachineHeating EXTENDS FB_SystemContinous
VAR_INPUT
END_VAR
VAR_OUTPUT
END_VAR
VAR
	//default parameters
	localDefaultParameters : ST_HNHT_CentralMachineHeatingDefaultParameters;
	
	//pumps
	stPU300DefaultParameters : ST_PumpGrundfosMagna3DefaultParameters := (tTaskCycleTime := GlobalVariables.tTaskCycleTime_MAIN, tCtrlCycleTime := GlobalVariables.tCtrlCycleTime_MAIN);
	PU300 : FB_PumpGrundfosMagna3 := (ST_DefaultParameters := stPU300DefaultParameters);;

	//valves
	stSV300DefaultParameters : ST_DiscreteValveDefaultParameters := (nFeedback := 0);
	SV300 : FB_DiscreteValve := (ST_DefaultParameters := stSV300DefaultParameters);
	
	//heat counter
	WMZ300: FB_MollineEHeatCounter;
	
	//internal variables
	bSetStatusOn_PU300 : BOOL;
	bSetStatusOn_SV300 : BOOL;
	
	bStartTimer : BOOL;
	Timer : TON;
END_VAR

MAIN();
//use timer because valve has no feedback signal (75 sec)
Timer(IN := bStartTimer,
	PT := T#75S);

SV300.GetState_BI();
SV300(bSetStatusOnAutomatic := bSetStatusOn_SV300,
	bAlgorithmPermission := bAlgorithmPermission);
SV300.SetState_BO();

PU300.GetState_Profibus();
PU300(bSetStatusOnAutomatic := bSetStatusOn_PU300,
	bAlgorithmPermission := bAlgorithmPermission,
	fThermalPowerExternal := WMZ300.fHeatFlowRate,
	fSetPointAutomatic := fSetPoint,
	nControlModeAutomatic := 3);
PU300.SetState_Profibus();

WMZ300(aHeatCounterTelegramm:=aTelegramm_WMZ300);

METHOD PROTECTED  CheckError : BOOL
VAR_INPUT
END_VAR
VAR_OUTPUT
	bError : BOOL;
END_VAR
IF PU300.bError THEN
	bError := TRUE;
END_IF
END_METHOD

METHOD PROTECTED  Operational : BOOL
VAR_INPUT
END_VAR
VAR_OUTPUT
	bSwitchToWorking : BOOL := FALSE;
END_VAR
bSetStatusOn_PU300 := TRUE;

IF PU300.bStatusOn THEN
	bSwitchToWorking := TRUE;
END_IF
END_METHOD

METHOD PROTECTED  RampDown : BOOL
VAR_INPUT
END_VAR
VAR_OUTPUT
	bRampDownFinished : BOOL := FALSE;
END_VAR
bSetStatusOn_PU300 := FALSE;

IF NOT PU300.bStatusOn THEN
	bSetStatusOn_SV300 := FALSE;
	bStartTimer := TRUE;
	IF Timer.Q THEN
		bRampDownFinished := TRUE;
		bStartTimer := FALSE;
	END_IF
END_IF
END_METHOD

METHOD PROTECTED  RampUp : BOOL
VAR_INPUT
END_VAR
VAR_OUTPUT
	bRampUpFinished : BOOL := FALSE;
END_VAR
bSetStatusOn_SV300 := TRUE;
bStartTimer := TRUE;

IF Timer.Q THEN
	bRampUpFinished := TRUE;
	bStartTimer := FALSE;
END_IF
END_METHOD

METHOD PROTECTED   SetSetPointLimits : BOOL
VAR_INPUT
END_VAR
IF  PU300.nControlModeAutomatic = 3 THEN
	aSetPointLimits[1] := localDefaultParameters.aSetPointLimitsTemperatureDifference[1];
	aSetPointLimits[2] := localDefaultParameters.aSetPointLimitsTemperatureDifference[2];
ELSE
	aSetPointLimits[1] := localDefaultParameters.aSetPointLimitsRelativeSpeed[1];
	aSetPointLimits[2] := localDefaultParameters.aSetPointLimitsRelativeSpeed[2];
END_IF
END_METHOD

METHOD PROTECTED  SetState : BOOL
VAR_INPUT
END_VAR
VAR_OUTPUT
END_VAR
fOperatingPoint := PU300.localState.fTemperatureDifference;

controlState.bStatusOn := bSetStatusOn;
setPointState.aSetPointLimits := aSetPointLimits;
setPointState.fSetPoint := fSetPoint;
setPointState.fOperatingPoint := fOperatingPoint;
setPointState.sSetPointUnit := 'K';
setPointState.sOperatingPointUnit := 'K';
END_METHOD

METHOD PROTECTED  Working : BOOL
VAR_INPUT
END_VAR
VAR_OUTPUT
	bSwitchToOperational : BOOL := FALSE;
END_VAR
//empty method
END_METHOD

END_FUNCTION_BLOCK

// ---- POUs/04 Systems/ConsumerSystems/HNHT/FB_AnnealingOvenExhaustGasSystem.TcPOU
FUNCTION_BLOCK FB_AnnealingOvenExhaustGasSystem EXTENDS FB_SystemContinous
VAR_INPUT
END_VAR
VAR_OUTPUT
END_VAR
VAR
	//default parameters
	localDefaultParameters : ST_AnnealingOvenExhaustGasDefaultParameters;

	//pumps
	stPU361DefaultParameters : ST_PumpGrundfosMagna3DefaultParameters := (bPumpBeforeApplication := FALSE, tTaskCycleTime := GlobalVariables.tTaskCycleTime_MAIN, tCtrlCycleTime := GlobalVariables.tCtrlCycleTime_MAIN);
	PU361 : FB_PumpGrundfosMagna3 := (ST_DefaultParameters := stPU361DefaultParameters);

	//valves
	stRV361DefaultParameters : ST_MixingValveDefaultParameters := (bFeedbackSignal := TRUE, tTaskCycleTime := GlobalVariables.tCtrlCycleTime_MAIN, tCtrlCycleTime := GlobalVariables.tCtrlCycleTime_MAIN, fOffsetTerminal := 7970);
	RV361 : FB_MixingValve := (ST_DefaultParameters := stRV361DefaultParameters);
	
	//heat counter	
	WMZ361 : FB_MollineC3HeatCounter;
	GM361 : FB_EmonioP3;
	
	//internal variables
	bSetStatusOn_PU361 : BOOL;
	bSetStatusOn_RV361 : BOOL;
END_VAR

MAIN();

//pumps
PU361.GetState_Profibus();
PU361(bSetStatusOnAutomatic := bSetStatusOn_PU361,
	fSetPointAutomatic := 100,
	bAlgorithmPermission := bAlgorithmPermission,
	nControlModeAutomatic := 0);
PU361.SetState_Profibus();

//valves
RV361.GetState_AI();
RV361(bSetStatusOnAutomatic := bSetStatusOn_RV361,
	fSetPointAutomatic := fSetPoint,
	bAlgorithmPermission := bAlgorithmPermission,
	fTemperatureExternal := PU361.fTemperatureInternal,
	fThermalPowerExternal := WMZ361.fHeatFlowRate,
	nControlModeAutomatic := 2);
RV361.SetState_AO();

WMZ361(aHeatCounterTelegramm := Telegramm_WZ_Abwaerme_Ofen_Abgasfackel);
GM361(sIPAddr := GlobalVariables.sIP_Emonio_AnnealingOven);

METHOD PROTECTED  CheckError : BOOL
VAR_INPUT
END_VAR
VAR_OUTPUT
	bError : BOOL;
END_VAR
bError := PU361.bError;
END_METHOD

METHOD PROTECTED  Operational : BOOL
VAR_INPUT
END_VAR
VAR_OUTPUT
	bSwitchToWorking : BOOL := FALSE;
END_VAR
bSetStatusOn_PU361 := TRUE;

IF PU361.bStatusOn THEN
	bSwitchToWorking := TRUE;
END_IF
END_METHOD

METHOD PROTECTED  RampDown : BOOL
VAR_INPUT
END_VAR
VAR_OUTPUT
	bRampDownFinished : BOOL := FALSE;
END_VAR
bSetStatusOn_PU361 := FALSE;

IF NOT PU361.bStatusOn THEN
	bSetStatusOn_RV361 := FALSE;
	IF RV361.fOperatingPoint<10 THEN
		bRampDownFinished := TRUE;
	END_IF
END_IF
END_METHOD

METHOD PROTECTED  RampUp : BOOL
VAR_INPUT
END_VAR
VAR_OUTPUT
	bRampUpFinished : BOOL := FALSE;
END_VAR
bSetStatusOn_RV361 := TRUE;
bRampUpFinished := TRUE;
END_METHOD

METHOD PROTECTED   SetSetPointLimits : BOOL
VAR_INPUT
END_VAR
aSetPointLimits[1] := localDefaultParameters.aSetPointLimitsTemperature[1];
aSetPointLimits[2] := localDefaultParameters.aSetPointLimitsTemperature[2];
END_METHOD

METHOD PROTECTED  SetState : BOOL
VAR_INPUT
END_VAR
VAR_OUTPUT
END_VAR
fOperatingPoint := PU361.fTemperatureInternal;

controlState.bStatusOn := bSetStatusOn;
setPointState.aSetPointLimits := aSetPointLimits;
setPointState.fSetPoint := fSetPoint;
setPointState.fOperatingPoint := fOperatingPoint;
setPointState.sSetPointUnit := 'degreeC';
setPointState.sOperatingPointUnit := 'degreeC';
END_METHOD

METHOD PROTECTED  Working : BOOL
VAR_INPUT
END_VAR
VAR_OUTPUT
	bSwitchToOperational : BOOL := FALSE;
END_VAR
//empty method
END_METHOD

END_FUNCTION_BLOCK

// ---- POUs/04 Systems/StorageSystems/FB_VSIStorageSystem.TcPOU
FUNCTION_BLOCK FB_VSIStorageSystem EXTENDS FB_SystemContinous
VAR_INPUT
	bLoadingAutomatic : BOOL; //variable to determine if storage is in loading mode
	fTemperatureBufferStorageSetPoint : REAL;
	fTemperatureBufferStorage : REAL;
END_VAR
VAR_OUTPUT
	localStorageState : ST_VSIStorageState;
END_VAR
VAR
	{attribute 'OPC.UA.DA' := '1'}
	localSetParameters : ST_ActiveStorageSystemSetParameters;
	{attribute 'OPC.UA.DA' := '1'}
	localState : ST_ActiveStorageSystemState;
	
	//default parameters
	localDefaultParameters : ST_VSIStorageSystemDefaultParameters;	

	//storage
	VSIStorage : FB_VSIStorage;
	
	//pumps
	
	stPU305DefaultParameters : ST_PumpGrundfosMagna3DefaultParameters := (bExternalTemperatureSensor := FALSE);
	PU305 : FB_PumpGrundfosMagna3 := (ST_DefaultParameters := stPU305DefaultParameters);; //Magna 3 pump (loading pump)
	PU306 : FB_PumpGrundfosMagna3 := (ST_DefaultParameters := stPU305DefaultParameters);; //Magna 3 pump (unloading pump)

	//valves
	stSV305DefaultParameters : ST_MixingValveDefaultParameters := (tTaskCycleTime := GlobalVariables.tTaskCycleTime_MAIN, tCtrlCycleTime := GlobalVariables.tCtrlCycleTime_MAIN, fOffsetTerminal := 4400);
	stSV306DefaultParameters : ST_MixingValveDefaultParameters := (tTaskCycleTime := GlobalVariables.tTaskCycleTime_MAIN, tCtrlCycleTime := GlobalVariables.tCtrlCycleTime_MAIN, fOffsetTerminal := 4400);
	stSV307DefaultParameters : ST_MixingValveDefaultParameters := (fControllerAmplification := 5, tControllerIntegralTime := T#500S, bARWOnIPartOnly := FALSE, tTaskCycleTime := GlobalVariables.tTaskCycleTime_MAIN, tCtrlCycleTime := GlobalVariables.tCtrlCycleTime_MAIN, fOutMinLimit := 25, fOffsetTerminal := 4400);
	
	SV305 : FB_MixingValve := (ST_DefaultParameters := stSV305DefaultParameters); //discrete inlet valve, valve motor needs continous signal but operates only between extreme positions
	SV306 : FB_MixingValve := (ST_DefaultParameters := stSV306DefaultParameters); //discrete outlet valve	, valve motor needs continous signal but operates only between extreme positions
	SV307 : FB_MixingValve := (ST_DefaultParameters := stSV307DefaultParameters); //discrete outlet valve	, valve motor needs continous signal but operates only between extreme positions
	
	WMZ305: FB_MollineEHeatCounter;
	
	//internal variables
	bSetStatusOn_PU305 : BOOL;
	bSetStatusOn_PU306 : BOOL;
	bSetStatusOn_SV305 : BOOL;
	fSetPoint_SV305 : REAL;
	bSetStatusOn_SV306 : BOOL;
	fSetPoint_SV306 : REAL;
	bSetStatusOn_SV307 : BOOL;
	fSetPoint_SV307 : REAL;
	fHeatFlowRate : REAL;
	bLoading : BOOL;
	nControlMode_SV307 : E_MixingValveControlMode; 
	
	//triggers
	SwitchToLoading : R_TRIG;
	SwitchToUnloading : F_TRIG;
	bFinishedSwitchMode : BOOL := TRUE;
END_VAR

//storage
VSIStorage(localState => localStorageState);

SelectLocalControlMode();
SwitchToLoading(CLK := bLoading);
SwitchToUnloading(CLK := bLoading);

//MAIN must be called before SwitchMode to prevent pump signal chattering (signal is written after SwitchMode function), SwitchMode may only be called if system is on
MAIN();

